(* Logix 5000 project; controller reports 1756-L63 rev 20.15; software revision 20.04 *)

TASK MainTask (continuous, watchdog 500 ms) : MainProgram, Report15Calcs, ReportCalcs

MODULES
   Local : 1756-L63 (ICP 0, rev 20.15)
END_MODULES

TYPE DateTime :
STRUCT
   Year : DINT;
   Month : DINT;
   Day : DINT;
   Hour : DINT;
   Minute : DINT;
   Second : DINT;
   Microsecond : DINT;   // Microsecond
   DayOfWeek : DINT;   // Day of week (Sunday = 0, Saturday = 6)
   DST_ON : BOOL;   // Day light Savings Time ON
END_STRUCT
END_TYPE

TYPE LogPoint :
STRUCT
   min : REAL;
   max : REAL;
   total : REAL;
   time : REAL;
   minminute : DINT;
   maxminute : DINT;
   valid : BOOL;
END_STRUCT
END_TYPE

TYPE LogRecord :
STRUCT
   log_data : LogPoint[125];
   time : DateTime;
END_STRUCT
END_TYPE

TYPE LogRecord15 :
STRUCT
   log_data : LogPoint[20];
   time : DateTime;
END_STRUCT
END_TYPE

TYPE LogRecord5 :
STRUCT
   log_data : LogPoint[20];
   time : DateTime;
END_STRUCT
END_TYPE

TYPE MOTOR :
STRUCT
   fail_dlay : DINT;
   mode_dlay : DINT;
   start_dlay : DINT;
   auto : BOOL;
   stop_man : BOOL;
   start_man : BOOL;
   fail_reset : BOOL;
   remote : BOOL;
   permit : BOOL;
   stop_sts : BOOL;
   run_sts : BOOL;
   stop_auto : BOOL;
   start_auto : BOOL;
   stop_out : BOOL;
   start_out : BOOL;
   run_out : BOOL;
   fail : BOOL;
   runtime : REAL;
   log : BOOL;
   Gen_Alarm : BOOL;   // General Alarm
   runtime_f : REAL;
   runtime_i : DINT;
   fail_tonr : FBD_TIMER;
   start_os : FBD_ONESHOT;
   manual_mode_timer : FBD_TIMER;
END_STRUCT
END_TYPE

TYPE PRANALOG :
STRUCT
   MinEU : REAL;
   MaxEU : REAL;
   almdb : REAL;
   lag : REAL;
   calib : BOOL;
   hihilim : REAL;
   hilim : REAL;
   lolim : REAL;
   lololim : REAL;
   raw : REAL;
   hold : BOOL;
   calc : REAL;
   value : REAL;
   valid : BOOL;
   log : BOOL;
   hihiraw : BOOL;
   hiraw : BOOL;
   loraw : BOOL;
   loloraw : BOOL;
END_STRUCT
END_TYPE

VAR_GLOBAL   (* controller tags *)
   AIT501do : PRANALOG := (MaxEU := 10.0, hihilim := 10.0, hilim := 8.0, lolim := 0.5, lololim := 0.5, raw := 21.951172, calc := 0.021951173, value := 0.021951173, valid := 1, log := 1, loraw := 1, loloraw := 1);   // Aeration tank 1 DO
   AIT501ph : PRANALOG := (MaxEU := 14.0, hihilim := 8.5, hilim := 8.0, lolim := 6.5, lololim := 6.3, raw := 5438.2197, calc := 7.6135077, value := 7.6135077, valid := 1, log := 1);   // Aeration tank 1 pH
   AIT502do : PRANALOG := (MaxEU := 10.0, hihilim := 10.0, hilim := 8.0, lolim := 0.5, lololim := 0.3, raw := 9517.547, calc := 9.517547, value := 9.517547, valid := 1, log := 1, hiraw := 1);   // Aeration tank 2 DO
   AIT502ph : PRANALOG := (MaxEU := 14.0, hihilim := 8.5, hilim := 8.0, lolim := 6.5, lololim := 6.3, raw := 4820.0977, calc := 6.7481365, value := 6.7481365, valid := 1, log := 1);   // Aeration tank 2 pH
   B301 : MOTOR := (fail_dlay := 60, start_dlay := 3000, permit := 1, run_sts := 1, runtime := 22541.49, runtime_f := 0.48989543, runtime_i := 22541, fail_tonr.TimerEnable := 1, fail_tonr.PRE := 60000, fail_tonr.Reset := 1, manual_mode_timer.Reset := 1);   // Equalization blower 1
   B302 : MOTOR := (fail_dlay := 60, start_dlay := 3000, permit := 1, run_sts := 1, runtime := 22540.76, runtime_f := 0.7594519, runtime_i := 22540, fail_tonr.TimerEnable := 1, fail_tonr.PRE := 60000, fail_tonr.Reset := 1, manual_mode_timer.Reset := 1);   // Equalization blower 2
   B303 : MOTOR := (fail_dlay := 60, start_dlay := 3000, permit := 1, stop_sts := 1, runtime := 0.2709657, runtime_f := 0.2709657, fail_tonr.TimerEnable := 1, fail_tonr.PRE := 60000, fail_tonr.Reset := 1, manual_mode_timer.Reset := 1);   // Equalization blower 3
   B501 : MOTOR := (fail_dlay := 60, start_dlay := 3000, auto := 1, remote := 1, permit := 1, stop_sts := 1, runtime := 10393.742, runtime_f := 0.7422347, runtime_i := 10393, fail_tonr.TimerEnable := 1, fail_tonr.PRE := 60000, fail_tonr.Reset := 1, manual_mode_timer.Reset := 1);   // Aeration tank 1 blower 1
   B502 : MOTOR := (fail_dlay := 60, start_dlay := 3000, auto := 1, remote := 1, permit := 1, stop_sts := 1, runtime := 6931.7354, runtime_f := 0.7353562, runtime_i := 6931, fail_tonr.TimerEnable := 1, fail_tonr.PRE := 60000, fail_tonr.Reset := 1, manual_mode_timer.Reset := 1);   // Aeration tank standby blower
   B503 : MOTOR := (fail_dlay := 60, start_dlay := 3000, auto := 1, remote := 1, permit := 1, run_sts := 1, run_out := 1, runtime := 5280.543, runtime_f := 0.5429669, runtime_i := 5280, fail_tonr.TimerEnable := 1, fail_tonr.PRE := 60000, fail_tonr.Reset := 1, start_os.InputBit := 1, manual_mode_timer.Reset := 1);   // Aeration tank 2 blower 1
   B601 : MOTOR := (fail_dlay := 60, start_dlay := 3000, remote := 1, permit := 1, stop_sts := 1, runtime := 17313.322, runtime_f := 0.32298738, runtime_i := 17313, fail_tonr.TimerEnable := 1, fail_tonr.PRE := 60000, fail_tonr.Reset := 1, manual_mode_timer.Reset := 1);   // Membrane tank 1 blower
   B602 : MOTOR := (fail_dlay := 60, start_dlay := 3000, remote := 1, permit := 1, stop_sts := 1, runtime := 12808.301, runtime_f := 0.30105218, runtime_i := 12808, fail_tonr.TimerEnable := 1, fail_tonr.PRE := 60000, fail_tonr.Reset := 1, manual_mode_timer.Reset := 1);   // Membrane tank 2 blower
   B603 : MOTOR := (fail_dlay := 60, start_dlay := 3000, auto := 1, remote := 1, permit := 1, run_sts := 1, run_out := 1, runtime := 5284.875, runtime_f := 0.87495077, runtime_i := 5284, fail_tonr.TimerEnable := 1, fail_tonr.PRE := 60000, fail_tonr.Reset := 1, start_os.InputBit := 1, manual_mode_timer.Reset := 1);   // Membrane tank 3 blower
   B604 : MOTOR := (fail_dlay := 60, start_dlay := 3000, auto := 1, remote := 1, permit := 1, run_sts := 1, run_out := 1, runtime := 5284.831, runtime_f := 0.8312785, runtime_i := 5284, fail_tonr.TimerEnable := 1, fail_tonr.PRE := 60000, fail_tonr.Reset := 1, start_os.InputBit := 1, manual_mode_timer.Reset := 1);   // Membrane tank 4 blower
   B901 : MOTOR := (fail_dlay := 60, start_dlay := 3000, remote := 1, permit := 1, stop_sts := 1, runtime := 1391.3846, runtime_f := 0.38459536, runtime_i := 1391, fail_tonr.TimerEnable := 1, fail_tonr.PRE := 60000, fail_tonr.Reset := 1, manual_mode_timer.Reset := 1);   // Digester blower 1
   B902 : MOTOR := (fail_dlay := 60, start_dlay := 3000, auto := 1, remote := 1, permit := 1, run_sts := 1, run_out := 1, runtime := 6851.961, runtime_f := 0.9611715, runtime_i := 6851, fail_tonr.TimerEnable := 1, fail_tonr.PRE := 60000, fail_tonr.Reset := 1, start_os.InputBit := 1, manual_mode_timer.Reset := 1);   // Digester blower 2
   DIESEL : MOTOR := (fail_dlay := 60, start_dlay := 3000, remote := 1, permit := 1, stop_sts := 1, fail_tonr.TimerEnable := 1, fail_tonr.PRE := 60000, fail_tonr.Reset := 1, manual_mode_timer.Reset := 1);   // Diesel generator
   FIT201 : PRANALOG := (MaxEU := 20.0, hihilim := 25.0, hilim := 20.0, raw := 3597.2026, calc := 7.194405, value := 7.194405, valid := 1, log := 1);   // Plant influent flow to screens
   FIT701 : PRANALOG := (MaxEU := 5.0, hihilim := 2.5, hilim := 2.0, lolim := 0.1, lololim := 0.1, raw := -9.0, valid := 1, log := 1, loraw := 1, loloraw := 1);   // Membrane tank 1 permeate flow
   FIT702 : PRANALOG := (MaxEU := 5.0, hihilim := 2.0, hilim := 1.8, lolim := 0.1, lololim := 0.1, raw := -4.0, valid := 1, log := 1, loraw := 1, loloraw := 1);   // Membrane tank 2 permeate flow
   FIT703 : PRANALOG := (MaxEU := 5.0, hihilim := 2.5, hilim := 2.0, lolim := 0.1, lololim := 0.1, raw := -4.0, valid := 1, log := 1, loraw := 1, loloraw := 1);   // Membrane tank 3 permeate flow
   FIT704 : PRANALOG := (MaxEU := 5.0, hihilim := 2.5, hilim := 2.0, raw := -6.0, valid := 1, log := 1);   // Membrane tank 4 permeate flow
   FIT801 : PRANALOG := (MaxEU := 5.0, raw := -1.0, valid := 1, log := 1, hihiraw := 1, hiraw := 1);   // CIP flow
   FIT901 : PRANALOG := (MaxEU := 5.0, raw := -4.0, valid := 1, log := 1, hihiraw := 1, hiraw := 1);   // Membrane tanks 1 & 2 WAS flow
   FIT902 : PRANALOG := (MaxEU := 5.0, raw := -3.0, valid := 1, log := 1, hihiraw := 1, hiraw := 1);   // Membrane tanks 3 & 4 WAS flow
   FunctionBlock_Cycle_Time : REAL := 251.0;   // Main Task Cycle Time in mseconds
   GT7951 : PRANALOG := (hihilim := 12.0, hilim := 10.0, raw := 125.78931, valid := 1, log := 1);   // Screening area H2S monitor
   LIT302 : PRANALOG := (MaxEU := 6.0, hihilim := 3.0, hilim := 2.9, lolim := 0.2, lololim := 0.5, raw := 1689.8391, calc := 1.0139034, value := 1.0139034, valid := 1, log := 1);   // Equalization tank 302 Level
   LIT501 : PRANALOG := (MaxEU := 6.0, hihilim := 2.5, hilim := 3.0, lolim := 1.0, lololim := 1.5, raw := 3821.76, calc := 2.293056, value := 2.293056, valid := 1, log := 1);   // Aeration tank 1 Level
   LIT502 : PRANALOG := (MaxEU := 6.0, hihilim := 2.5, hilim := 3.0, lolim := 1.0, lololim := 1.5, raw := 3509.0679, calc := 2.1054406, value := 2.1054406, valid := 1, log := 1);   // Aeration tank 2 Level
   LIT6101 : PRANALOG := (MaxEU := 2.0, raw := 795.14307, calc := 0.15902862, value := 0.15902862, valid := 1, log := 1, hihiraw := 1, hiraw := 1);   // Coagulant tank 6101 level
   LIT6102 : PRANALOG := (MaxEU := 2.0, raw := 931.36914, calc := 0.18627383, value := 0.18627383, valid := 1, log := 1, hihiraw := 1, hiraw := 1);   // Caustic tank 6102 Leve
   P301 : MOTOR := (fail_dlay := 60, start_dlay := 3000, remote := 1, permit := 1, stop_sts := 1, runtime := 502.63425, runtime_f := 0.6342328, runtime_i := 502, fail_tonr.TimerEnable := 1, fail_tonr.PRE := 60000, fail_tonr.Reset := 1, manual_mode_timer.Reset := 1);   // Equalization pump 1
   P302 : MOTOR := (fail_dlay := 60, start_dlay := 3000, remote := 1, permit := 1, stop_sts := 1, runtime := 1.2261261, runtime_f := 0.22612606, runtime_i := 1, fail_tonr.TimerEnable := 1, fail_tonr.PRE := 60000, fail_tonr.Reset := 1, manual_mode_timer.Reset := 1);   // Equalization pump 2
   P303 : MOTOR := (fail_dlay := 60, start_dlay := 3000, auto := 1, remote := 1, permit := 1, stop_sts := 1, runtime := 201.53206, runtime_f := 0.5320589, runtime_i := 201, fail_tonr.TimerEnable := 1, fail_tonr.PRE := 60000, fail_tonr.Reset := 1, manual_mode_timer.Reset := 1);   // Equalization pump 3
   P501 : MOTOR := (fail_dlay := 60, start_dlay := 3000, remote := 1, permit := 1, stop_sts := 1, runtime := 14554.279, runtime_f := 0.27947924, runtime_i := 14554, fail_tonr.TimerEnable := 1, fail_tonr.PRE := 60000, fail_tonr.Reset := 1, manual_mode_timer.Reset := 1);   // Membrane tank 1 mixed liquor pump
   P502 : MOTOR := (fail_dlay := 60, start_dlay := 3000, remote := 1, permit := 1, stop_sts := 1, runtime := 11217.086, runtime_f := 0.08595178, runtime_i := 11217, fail_tonr.TimerEnable := 1, fail_tonr.PRE := 60000, fail_tonr.Reset := 1, manual_mode_timer.Reset := 1);   // Membrane tank 2 mixed liquor pump
   P503 : MOTOR := (fail_dlay := 60, start_dlay := 3000, auto := 1, remote := 1, permit := 1, stop_sts := 1, runtime := 4799.387, runtime_f := 0.38708004, runtime_i := 4799, fail_tonr.TimerEnable := 1, fail_tonr.PRE := 60000, fail_tonr.Reset := 1, manual_mode_timer.Reset := 1);   // Membrane tank 3 mixed liquor pump
   P504 : MOTOR := (fail_dlay := 60, start_dlay := 3000, auto := 1, remote := 1, permit := 1, stop_sts := 1, runtime := 4738.982, runtime_f := 0.98173386, runtime_i := 4738, fail_tonr.TimerEnable := 1, fail_tonr.PRE := 60000, fail_tonr.Reset := 1, manual_mode_timer.Reset := 1);   // Membrane tank 4 mixed liquor pump
   P7011 : MOTOR := (fail_dlay := 60, start_dlay := 3000, auto := 1, remote := 1, permit := 1, stop_sts := 1, runtime := 6253.749, runtime_f := 0.7490861, runtime_i := 6253, fail_tonr.TimerEnable := 1, fail_tonr.PRE := 60000, fail_tonr.Reset := 1, manual_mode_timer.Reset := 1);   // Membrane tank 1 permeate pump 1
   P7012 : MOTOR := (fail_dlay := 60, start_dlay := 3000, auto := 1, remote := 1, permit := 1, stop_sts := 1, runtime := 5870.5024, runtime_f := 0.502557, runtime_i := 5870, fail_tonr.TimerEnable := 1, fail_tonr.PRE := 60000, fail_tonr.Reset := 1, manual_mode_timer.Reset := 1);   // Membrane tank 1 permeate pump 2
   P7021 : MOTOR := (fail_dlay := 60, start_dlay := 3000, auto := 1, remote := 1, permit := 1, stop_sts := 1, runtime := 4789.597, runtime_f := 0.59710574, runtime_i := 4789, fail_tonr.TimerEnable := 1, fail_tonr.PRE := 60000, fail_tonr.Reset := 1, manual_mode_timer.Reset := 1);   // Membrane tank 2 permeate pump 1
   P7022 : MOTOR := (fail_dlay := 60, start_dlay := 3000, auto := 1, remote := 1, permit := 1, stop_sts := 1, runtime := 4792.9336, runtime_f := 0.9336782, runtime_i := 4792, fail_tonr.TimerEnable := 1, fail_tonr.PRE := 60000, fail_tonr.Reset := 1, manual_mode_timer.Reset := 1);   // Membrane tank 2 permeate pump 2
   P7031 : MOTOR := (fail_dlay := 60, start_dlay := 3000, auto := 1, remote := 1, permit := 1, stop_sts := 1, runtime := 2042.6858, runtime_f := 0.6858263, runtime_i := 2042, fail_tonr.TimerEnable := 1, fail_tonr.PRE := 60000, fail_tonr.Reset := 1, manual_mode_timer.Reset := 1);   // Membrane tank 3 permeate pump 1
   P7032 : MOTOR := (fail_dlay := 60, start_dlay := 3000, auto := 1, remote := 1, permit := 1, stop_sts := 1, runtime := 2005.9248, runtime_f := 0.924792, runtime_i := 2005, fail_tonr.TimerEnable := 1, fail_tonr.PRE := 60000, fail_tonr.Reset := 1, manual_mode_timer.Reset := 1);   // Membrane tank 3 permeate pump 2
   P7041 : MOTOR := (fail_dlay := 60, start_dlay := 3000, auto := 1, remote := 1, permit := 1, stop_sts := 1, runtime := 1973.3212, runtime_f := 0.32117462, runtime_i := 1973, fail_tonr.TimerEnable := 1, fail_tonr.PRE := 60000, fail_tonr.Reset := 1, manual_mode_timer.Reset := 1);   // Membrane tank 4 permeate pump 1
   P7042 : MOTOR := (fail_dlay := 60, start_dlay := 3000, auto := 1, remote := 1, permit := 1, stop_sts := 1, runtime := 1973.0812, runtime_f := 0.081213675, runtime_i := 1973, fail_tonr.TimerEnable := 1, fail_tonr.PRE := 60000, fail_tonr.Reset := 1, manual_mode_timer.Reset := 1);   // Membrane tank 4 permeate pump 2
   P7951 : MOTOR := (permit := 1, stop_sts := 1, fail_tonr.TimerEnable := 1, fail_tonr.Reset := 1, manual_mode_timer.Reset := 1);   // Screen building sump pump
   P801 : MOTOR := (fail_dlay := 60, start_dlay := 3000, auto := 1, remote := 1, permit := 1, stop_sts := 1, runtime := 62.99539, runtime_f := 0.9953907, runtime_i := 62, fail_tonr.TimerEnable := 1, fail_tonr.PRE := 60000, fail_tonr.Reset := 1, manual_mode_timer.Reset := 1);   // CIP pump 1
   P802 : MOTOR := (fail_dlay := 60, auto := 1, remote := 1, permit := 1, stop_sts := 1, runtime := 411.53458, runtime_f := 0.5345711, runtime_i := 411, fail_tonr.TimerEnable := 1, fail_tonr.PRE := 60000, fail_tonr.Reset := 1, manual_mode_timer.Reset := 1);   // CIP Pump 2
   P901 : MOTOR := (fail_dlay := 60, start_dlay := 3000, remote := 1, permit := 1, stop_sts := 1, runtime := 70.41078, runtime_f := 0.4107828, runtime_i := 70, fail_tonr.TimerEnable := 1, fail_tonr.PRE := 60000, fail_tonr.Reset := 1, manual_mode_timer.Reset := 1);   // Membrane tank 1 WAS pump
   P902 : MOTOR := (fail_dlay := 60, start_dlay := 3000, remote := 1, permit := 1, stop_sts := 1, runtime := 51.641758, runtime_f := 0.6417567, runtime_i := 51, fail_tonr.TimerEnable := 1, fail_tonr.PRE := 60000, fail_tonr.Reset := 1, manual_mode_timer.Reset := 1);   // Membrane tank 2 WAS pump
   P903 : MOTOR := (fail_dlay := 60, start_dlay := 3000, remote := 1, permit := 1, run_sts := 1, run_out := 1, runtime := 14599.742, runtime_f := 0.7419928, runtime_i := 14599, fail_tonr.TimerEnable := 1, fail_tonr.PRE := 60000, fail_tonr.Reset := 1, start_os.InputBit := 1, manual_mode_timer.Reset := 1);   // Digester decant pump
   P904 : MOTOR := (fail_dlay := 60, start_dlay := 3000, remote := 1, permit := 1, stop_sts := 1, runtime := 23.586103, runtime_f := 0.58610374, runtime_i := 23, fail_tonr.TimerEnable := 1, fail_tonr.PRE := 60000, fail_tonr.Reset := 1, manual_mode_timer.Reset := 1);   // Membrane tank 4 WAS pump
   P905 : MOTOR := (fail_dlay := 60, start_dlay := 3000, remote := 1, permit := 1, stop_sts := 1, runtime := 22.263817, runtime_f := 0.26381716, runtime_i := 22, fail_tonr.TimerEnable := 1, fail_tonr.PRE := 60000, fail_tonr.Reset := 1, manual_mode_timer.Reset := 1);   // Membrane tank 3 WAS pump
   report15_data : LogRecord15[800] := ([0].log_data[0].min := 1.0, [0].log_data[0].max := 1.0, [0].log_data[0].total := 900.0, [0].log_data[0].time := 900.0, [0].log_data[0].minminute := 15, [0].log_data[0].maxminute := 15, [0].log_data[0].valid := 1, [0].log_data[1].valid := 1, [0].log_data[2].valid := 1, [0].log_data[3].valid := 1, [0].log_data[4].valid := 1, [0].log_data[5].valid := 1, [0].log_data[6].valid := 1, [0].log_data[7].valid := 1, [0].log_data[8].valid := 1, [0].log_data[9].valid := 1, [0].log_data[10].valid := 1, [0].log_data[11].valid := 1, [0].log_data[12].valid := 1, [0].log_data[13].valid := 1, [0].log_data[14].valid := 1, [0].log_data[15].valid := 1, [0].log_data[16].valid := 1, [0].log_data[17].valid := 1, [0].log_data[18].valid := 1, [0].log_data[19].valid := 1, [0].time.Year := 2023, [0].time.Month := 1, [0].time.Day := 16, [0].time.Minute := 29, [0].time.Second := 59, [1].log_data[0].min := 1.0, [1].log_data[0].max := 1.0, [1].log_data[0].total := 900.0, [1].log_data[0].time := 900.0, [1].log_data[0].minminute := 30, [1].log_data[0].maxminute := 30, [1].log_data[0].valid := 1, [1].log_data[1].valid := 1, [1].log_data[2].valid := 1, [1].log_data[3].valid := 1, [1].log_data[4].valid := 1, [1].log_data[5].valid := 1, [1].log_data[6].valid := 1, [1].log_data[7].valid := 1, [1].log_data[8].valid := 1, [1].log_data[9].valid := 1, [1].log_data[10].valid := 1, [1].log_data[11].valid := 1, [1].log_data[12].valid := 1, [1].log_data[13].valid := 1, [1].log_data[14].valid := 1, [1].log_data[15].valid := 1, [1].log_data[16].valid := 1, [1].log_data[17].valid := 1, [1].log_data[18].valid := 1, [1].log_data[19].valid := 1, [1].time.Year := 2023, [1].time.Month := 1, [1].time.Day := 16,
        [1].time.Minute := 44, [1].time.Second := 59, [2].log_data[0].min := 1.0, [2].log_data[0].max := 1.0, [2].log_data[0].total := 900.0, [2].log_data[0].time := 900.0, [2].log_data[0].minminute := 45, [2].log_data[0].maxminute := 45, [2].log_data[0].valid := 1, [2].log_data[1].valid := 1, [2].log_data[2].valid := 1, [2].log_data[3].valid := 1, [2].log_data[4].valid := 1, [2].log_data[5].valid := 1, [2].log_data[6].valid := 1, [2].log_data[7].valid := 1, [2].log_data[8].valid := 1, [2].log_data[9].valid := 1, [2].log_data[10].valid := 1, [2].log_data[11].valid := 1, [2].log_data[12].valid := 1, [2].log_data[13].valid := 1, [2].log_data[14].valid := 1, [2].log_data[15].valid := 1, [2].log_data[16].valid := 1, [2].log_data[17].valid := 1, [2].log_data[18].valid := 1, [2].log_data[19].valid := 1, [2].time.Year := 2023, [2].time.Month := 1, [2].time.Day := 16, [2].time.Minute := 59, [2].time.Second := 59, [3].log_data[0].min := 1.0, [3].log_data[0].max := 1.0, [3].log_data[0].total := 900.0, [3].log_data[0].time := 900.0, [3].log_data[0].valid := 1, [3].log_data[1].valid := 1, [3].log_data[2].valid := 1, [3].log_data[3].valid := 1, [3].log_data[4].valid := 1, [3].log_data[5].valid := 1, [3].log_data[6].valid := 1, [3].log_data[7].valid := 1, [3].log_data[8].valid := 1, [3].log_data[9].valid := 1, [3].log_data[10].valid := 1, [3].log_data[11].valid := 1, [3].log_data[12].valid := 1, [3].log_data[13].valid := 1, [3].log_data[14].valid := 1, [3].log_data[15].valid := 1, [3].log_data[16].valid := 1, [3].log_data[17].valid := 1, [3].log_data[18].valid := 1, [3].log_data[19].valid := 1, [3].time.Year := 2023, [3].time.Month := 1, [3].time.Day := 16,
        [3].time.Hour := 1, [3].time.Minute := 14, [3].time.Second := 59, [4].log_data[0].min := 1.0, [4].log_data[0].max := 1.0, [4].log_data[0].total := 900.0, [4].log_data[0].time := 900.0, [4].log_data[0].minminute := 15, [4].log_data[0].maxminute := 15, [4].log_data[0].valid := 1, [4].log_data[1].valid := 1, [4].log_data[2].valid := 1, [4].log_data[3].valid := 1, [4].log_data[4].valid := 1, [4].log_data[5].valid := 1, [4].log_data[6].valid := 1, [4].log_data[7].valid := 1, [4].log_data[8].valid := 1, [4].log_data[9].valid := 1, [4].log_data[10].valid := 1, [4].log_data[11].valid := 1, [4].log_data[12].valid := 1, [4].log_data[13].valid := 1, [4].log_data[14].valid := 1, [4].log_data[15].valid := 1, [4].log_data[16].valid := 1, [4].log_data[17].valid := 1, [4].log_data[18].valid := 1, [4].log_data[19].valid := 1, [4].time.Year := 2023, [4].time.Month := 1, [4].time.Day := 16, [4].time.Hour := 1, [4].time.Minute := 29, [4].time.Second := 59, [5].log_data[0].min := 1.0, [5].log_data[0].max := 1.0, [5].log_data[0].total := 900.0, [5].log_data[0].time := 900.0, [5].log_data[0].minminute := 30, [5].log_data[0].maxminute := 30, [5].log_data[0].valid := 1, [5].log_data[1].valid := 1, [5].log_data[2].valid := 1, [5].log_data[3].valid := 1, [5].log_data[4].valid := 1, [5].log_data[5].valid := 1, [5].log_data[6].valid := 1, [5].log_data[7].valid := 1, [5].log_data[8].valid := 1, [5].log_data[9].valid := 1, [5].log_data[10].valid := 1, [5].log_data[11].valid := 1, [5].log_data[12].valid := 1, [5].log_data[13].valid := 1, [5].log_data[14].valid := 1, [5].log_data[15].valid := 1, [5].log_data[16].valid := 1, [5].log_data[17].valid := 1, [5].log_data[18].valid := 1,
        [5].log_data[19].valid := 1, [5].time.Year := 2023, [5].time.Month := 1, [5].time.Day := 16, [5].time.Hour := 1, [5].time.Minute := 44, [5].time.Second := 59, [6].log_data[0].min := 1.0, [6].log_data[0].max := 1.0, [6].log_data[0].total := 900.0, [6].log_data[0].time := 900.0, [6].log_data[0].minminute := 45, [6].log_data[0].maxminute := 45, [6].log_data[0].valid := 1, [6].log_data[1].valid := 1, [6].log_data[2].valid := 1, [6].log_data[3].valid := 1, [6].log_data[4].valid := 1, [6].log_data[5].valid := 1, [6].log_data[6].valid := 1, [6].log_data[7].valid := 1, [6].log_data[8].valid := 1, [6].log_data[9].valid := 1, [6].log_data[10].valid := 1, [6].log_data[11].valid := 1, [6].log_data[12].valid := 1, [6].log_data[13].valid := 1, [6].log_data[14].valid := 1, [6].log_data[15].valid := 1, [6].log_data[16].valid := 1, [6].log_data[17].valid := 1, [6].log_data[18].valid := 1, [6].log_data[19].valid := 1, [6].time.Year := 2023, [6].time.Month := 1, [6].time.Day := 16, [6].time.Hour := 1, [6].time.Minute := 59, [6].time.Second := 59, [7].log_data[0].min := 1.0, [7].log_data[0].max := 1.0, [7].log_data[0].total := 900.0, [7].log_data[0].time := 900.0, [7].log_data[0].valid := 1, [7].log_data[1].valid := 1, [7].log_data[2].valid := 1, [7].log_data[3].valid := 1, [7].log_data[4].valid := 1, [7].log_data[5].valid := 1, [7].log_data[6].valid := 1, [7].log_data[7].valid := 1, [7].log_data[8].valid := 1, [7].log_data[9].valid := 1, [7].log_data[10].valid := 1, [7].log_data[11].valid := 1, [7].log_data[12].valid := 1, [7].log_data[13].valid := 1, [7].log_data[14].valid := 1, [7].log_data[15].valid := 1, [7].log_data[16].valid := 1,
        [7].log_data[17].valid := 1, [7].log_data[18].valid := 1, [7].log_data[19].valid := 1, [7].time.Year := 2023, [7].time.Month := 1, [7].time.Day := 16, [7].time.Hour := 2, [7].time.Minute := 14, [7].time.Second := 59, [8].log_data[0].min := 1.0, [8].log_data[0].max := 1.0, [8].log_data[0].total := 900.0, [8].log_data[0].time := 900.0, [8].log_data[0].minminute := 15, [8].log_data[0].maxminute := 15, [8].log_data[0].valid := 1, [8].log_data[1].valid := 1, [8].log_data[2].valid := 1, [8].log_data[3].valid := 1, [8].log_data[4].valid := 1, [8].log_data[5].valid := 1, [8].log_data[6].valid := 1, [8].log_data[7].valid := 1, [8].log_data[8].valid := 1, [8].log_data[9].valid := 1, [8].log_data[10].valid := 1, [8].log_data[11].valid := 1, [8].log_data[12].valid := 1, [8].log_data[13].valid := 1, [8].log_data[14].valid := 1, [8].log_data[15].valid := 1, [8].log_data[16].valid := 1, [8].log_data[17].valid := 1, [8].log_data[18].valid := 1, [8].log_data[19].valid := 1, [8].time.Year := 2023, [8].time.Month := 1, [8].time.Day := 16, [8].time.Hour := 2, [8].time.Minute := 29, [8].time.Second := 59, [9].log_data[0].min := 1.0, [9].log_data[0].max := 1.0, [9].log_data[0].total := 900.0, [9].log_data[0].time := 900.0, [9].log_data[0].minminute := 30, [9].log_data[0].maxminute := 30, [9].log_data[0].valid := 1, [9].log_data[1].valid := 1, [9].log_data[2].valid := 1, [9].log_data[3].valid := 1, [9].log_data[4].valid := 1, [9].log_data[5].valid := 1, [9].log_data[6].valid := 1, [9].log_data[7].valid := 1, [9].log_data[8].valid := 1, [9].log_data[9].valid := 1, [9].log_data[10].valid := 1, [9].log_data[11].valid := 1, [9].log_data[12].valid := 1,
        [9].log_data[13].valid := 1, [9].log_data[14].valid := 1, [9].log_data[15].valid := 1, [9].log_data[16].valid := 1, [9].log_data[17].valid := 1, [9].log_data[18].valid := 1, [9].log_data[19].valid := 1, [9].time.Year := 2023, [9].time.Month := 1, [9].time.Day := 16, [9].time.Hour := 2, [9].time.Minute := 44, [9].time.Second := 59, [10].log_data[0].min := 1.0, [10].log_data[0].max := 1.0, [10].log_data[0].total := 900.0, [10].log_data[0].time := 900.0, [10].log_data[0].minminute := 45, [10].log_data[0].maxminute := 45, [10].log_data[0].valid := 1, [10].log_data[1].valid := 1, [10].log_data[2].valid := 1, [10].log_data[3].valid := 1, [10].log_data[4].valid := 1, [10].log_data[5].valid := 1, [10].log_data[6].valid := 1, [10].log_data[7].valid := 1, [10].log_data[8].valid := 1, [10].log_data[9].valid := 1, [10].log_data[10].valid := 1, [10].log_data[11].valid := 1, [10].log_data[12].valid := 1, [10].log_data[13].valid := 1, [10].log_data[14].valid := 1, [10].log_data[15].valid := 1, [10].log_data[16].valid := 1, [10].log_data[17].valid := 1, [10].log_data[18].valid := 1, [10].log_data[19].valid := 1, [10].time.Year := 2023, [10].time.Month := 1, [10].time.Day := 16, [10].time.Hour := 2, [10].time.Minute := 59, [10].time.Second := 59, [11].log_data[0].min := 1.0, [11].log_data[0].max := 1.0, [11].log_data[0].total := 900.0, [11].log_data[0].time := 900.0, [11].log_data[0].valid := 1, [11].log_data[1].valid := 1, [11].log_data[2].valid := 1, [11].log_data[3].valid := 1, [11].log_data[4].valid := 1, [11].log_data[5].valid := 1, [11].log_data[6].valid := 1, [11].log_data[7].valid := 1, [11].log_data[8].valid := 1, [11].log_data[9].valid := 1, [11].log_data[10].valid := 1,
        [11].log_data[11].valid := 1, [11].log_data[12].valid := 1, [11].log_data[13].valid := 1, [11].log_data[14].valid := 1, [11].log_data[15].valid := 1, [11].log_data[16].valid := 1, [11].log_data[17].valid := 1, [11].log_data[18].valid := 1, [11].log_data[19].valid := 1, [11].time.Year := 2023, [11].time.Month := 1, [11].time.Day := 16, [11].time.Hour := 3, [11].time.Minute := 14, [11].time.Second := 59, [12].log_data[0].min := 1.0, [12].log_data[0].max := 1.0, [12].log_data[0].total := 900.0, [12].log_data[0].time := 900.0, [12].log_data[0].minminute := 15, [12].log_data[0].maxminute := 15, [12].log_data[0].valid := 1, [12].log_data[1].valid := 1, [12].log_data[2].valid := 1, [12].log_data[3].valid := 1, [12].log_data[4].valid := 1, [12].log_data[5].valid := 1, [12].log_data[6].valid := 1, [12].log_data[7].valid := 1, [12].log_data[8].valid := 1, [12].log_data[9].valid := 1, [12].log_data[10].valid := 1, [12].log_data[11].valid := 1, [12].log_data[12].valid := 1, [12].log_data[13].valid := 1, [12].log_data[14].valid := 1, [12].log_data[15].valid := 1, [12].log_data[16].valid := 1, [12].log_data[17].valid := 1, [12].log_data[18].valid := 1, [12].log_data[19].valid := 1, [12].time.Year := 2023, [12].time.Month := 1, [12].time.Day := 16, [12].time.Hour := 3, [12].time.Minute := 29, [12].time.Second := 59, [13].log_data[0].min := 1.0, [13].log_data[0].max := 1.0, [13].log_data[0].total := 900.0, [13].log_data[0].time := 900.0, [13].log_data[0].minminute := 30, [13].log_data[0].maxminute := 30, [13].log_data[0].valid := 1, [13].log_data[1].valid := 1, [13].log_data[2].valid := 1, [13].log_data[3].valid := 1, [13].log_data[4].valid := 1, [13].log_data[5].valid := 1, [13].log_data[6].valid := 1,
        [13].log_data[7].valid := 1, [13].log_data[8].valid := 1, [13].log_data[9].valid := 1, [13].log_data[10].valid := 1, [13].log_data[11].valid := 1, [13].log_data[12].valid := 1, [13].log_data[13].valid := 1, [13].log_data[14].valid := 1, [13].log_data[15].valid := 1, [13].log_data[16].valid := 1, [13].log_data[17].valid := 1, [13].log_data[18].valid := 1, [13].log_data[19].valid := 1, [13].time.Year := 2023, [13].time.Month := 1, [13].time.Day := 16, [13].time.Hour := 3, [13].time.Minute := 44, [13].time.Second := 59, [14].log_data[0].min := 1.0, [14].log_data[0].max := 1.0, [14].log_data[0].total := 900.0, [14].log_data[0].time := 900.0, [14].log_data[0].minminute := 45, [14].log_data[0].maxminute := 45, [14].log_data[0].valid := 1, [14].log_data[1].valid := 1, [14].log_data[2].valid := 1, [14].log_data[3].valid := 1, [14].log_data[4].valid := 1, [14].log_data[5].valid := 1, [14].log_data[6].valid := 1, [14].log_data[7].valid := 1, [14].log_data[8].valid := 1, [14].log_data[9].valid := 1, [14].log_data[10].valid := 1, [14].log_data[11].valid := 1, [14].log_data[12].valid := 1, [14].log_data[13].valid := 1, [14].log_data[14].valid := 1, [14].log_data[15].valid := 1, [14].log_data[16].valid := 1, [14].log_data[17].valid := 1, [14].log_data[18].valid := 1, [14].log_data[19].valid := 1, [14].time.Year := 2023, [14].time.Month := 1, [14].time.Day := 16, [14].time.Hour := 3, [14].time.Minute := 59, [14].time.Second := 59, [15].log_data[0].min := 1.0, [15].log_data[0].max := 1.0, [15].log_data[0].total := 900.0, [15].log_data[0].time := 900.0, [15].log_data[0].valid := 1, [15].log_data[1].valid := 1, [15].log_data[2].valid := 1, [15].log_data[3].valid := 1, [15].log_data[4].valid := 1,
        [15].log_data[5].valid := 1, [15].log_data[6].valid := 1, [15].log_data[7].valid := 1, [15].log_data[8].valid := 1, [15].log_data[9].valid := 1, [15].log_data[10].valid := 1, [15].log_data[11].valid := 1, [15].log_data[12].valid := 1, [15].log_data[13].valid := 1, [15].log_data[14].valid := 1, [15].log_data[15].valid := 1, [15].log_data[16].valid := 1, [15].log_data[17].valid := 1, [15].log_data[18].valid := 1, [15].log_data[19].valid := 1, [15].time.Year := 2023, [15].time.Month := 1, [15].time.Day := 16, [15].time.Hour := 4, [15].time.Minute := 14, [15].time.Second := 59, [16].log_data[0].min := 1.0, [16].log_data[0].max := 1.0, [16].log_data[0].total := 900.0, [16].log_data[0].time := 900.0, [16].log_data[0].minminute := 15, [16].log_data[0].maxminute := 15, [16].log_data[0].valid := 1, [16].log_data[1].valid := 1, [16].log_data[2].valid := 1, [16].log_data[3].valid := 1, [16].log_data[4].valid := 1, [16].log_data[5].valid := 1, [16].log_data[6].valid := 1, [16].log_data[7].valid := 1, [16].log_data[8].valid := 1, [16].log_data[9].valid := 1, [16].log_data[10].valid := 1, [16].log_data[11].valid := 1, [16].log_data[12].valid := 1, [16].log_data[13].valid := 1, [16].log_data[14].valid := 1, [16].log_data[15].valid := 1, [16].log_data[16].valid := 1, [16].log_data[17].valid := 1, [16].log_data[18].valid := 1, [16].log_data[19].valid := 1, [16].time.Year := 2023, [16].time.Month := 1, [16].time.Day := 16, [16].time.Hour := 4, [16].time.Minute := 29, [16].time.Second := 59, [17].log_data[0].min := 1.0, [17].log_data[0].max := 1.0, [17].log_data[0].total := 900.0, [17].log_data[0].time := 900.0, [17].log_data[0].minminute := 30, [17].log_data[0].maxminute := 30, [17].log_data[0].valid := 1,
        [17].log_data[1].valid := 1, [17].log_data[2].valid := 1, [17].log_data[3].valid := 1, [17].log_data[4].valid := 1, [17].log_data[5].valid := 1, [17].log_data[6].valid := 1, [17].log_data[7].valid := 1, [17].log_data[8].valid := 1, [17].log_data[9].valid := 1, [17].log_data[10].valid := 1, [17].log_data[11].valid := 1, [17].log_data[12].valid := 1, [17].log_data[13].valid := 1, [17].log_data[14].valid := 1, [17].log_data[15].valid := 1, [17].log_data[16].valid := 1, [17].log_data[17].valid := 1, [17].log_data[18].valid := 1, [17].log_data[19].valid := 1, [17].time.Year := 2023, [17].time.Month := 1, [17].time.Day := 16, [17].time.Hour := 4, [17].time.Minute := 44, [17].time.Second := 59, [18].log_data[0].min := 1.0, [18].log_data[0].max := 1.0, [18].log_data[0].total := 900.0, [18].log_data[0].time := 900.0, [18].log_data[0].minminute := 45, [18].log_data[0].maxminute := 45, [18].log_data[0].valid := 1, [18].log_data[1].valid := 1, [18].log_data[2].valid := 1, [18].log_data[3].valid := 1, [18].log_data[4].valid := 1, [18].log_data[5].valid := 1, [18].log_data[6].valid := 1, [18].log_data[7].valid := 1, [18].log_data[8].valid := 1, [18].log_data[9].valid := 1, [18].log_data[10].valid := 1, [18].log_data[11].valid := 1, [18].log_data[12].valid := 1, [18].log_data[13].valid := 1, [18].log_data[14].valid := 1, [18].log_data[15].valid := 1, [18].log_data[16].valid := 1, [18].log_data[17].valid := 1, [18].log_data[18].valid := 1, [18].log_data[19].valid := 1, [18].time.Year := 2023, [18].time.Month := 1, [18].time.Day := 16, [18].time.Hour := 4, [18].time.Minute := 59, [18].time.Second := 59, [19].log_data[0].min := 1.0, [19].log_data[0].max := 1.0, [19].log_data[0].total := 900.0,
        [19].log_data[0].time := 900.0, [19].log_data[0].valid := 1, [19].log_data[1].valid := 1, [19].log_data[2].valid := 1, [19].log_data[3].valid := 1, [19].log_data[4].valid := 1, [19].log_data[5].valid := 1, [19].log_data[6].valid := 1, [19].log_data[7].valid := 1, [19].log_data[8].valid := 1, [19].log_data[9].valid := 1, [19].log_data[10].valid := 1, [19].log_data[11].valid := 1, [19].log_data[12].valid := 1, [19].log_data[13].valid := 1, [19].log_data[14].valid := 1, [19].log_data[15].valid := 1, [19].log_data[16].valid := 1, [19].log_data[17].valid := 1, [19].log_data[18].valid := 1, [19].log_data[19].valid := 1, [19].time.Year := 2023, [19].time.Month := 1, [19].time.Day := 16, [19].time.Hour := 5, [19].time.Minute := 14, [19].time.Second := 59, [20].log_data[0].min := 1.0, [20].log_data[0].max := 1.0, [20].log_data[0].total := 900.0, [20].log_data[0].time := 900.0, [20].log_data[0].minminute := 15, [20].log_data[0].maxminute := 15, [20].log_data[0].valid := 1, [20].log_data[1].valid := 1, [20].log_data[2].valid := 1, [20].log_data[3].valid := 1, [20].log_data[4].valid := 1, [20].log_data[5].valid := 1, [20].log_data[6].valid := 1, [20].log_data[7].valid := 1, [20].log_data[8].valid := 1, [20].log_data[9].valid := 1, [20].log_data[10].valid := 1, [20].log_data[11].valid := 1, [20].log_data[12].valid := 1, [20].log_data[13].valid := 1, [20].log_data[14].valid := 1, [20].log_data[15].valid := 1, [20].log_data[16].valid := 1, [20].log_data[17].valid := 1, [20].log_data[18].valid := 1, [20].log_data[19].valid := 1, [20].time.Year := 2023, [20].time.Month := 1, [20].time.Day := 16, [20].time.Hour := 5, [20].time.Minute := 29, [20].time.Second := 59, [21].log_data[0].min := 1.0,
        [21].log_data[0].max := 1.0, [21].log_data[0].total := 900.0, [21].log_data[0].time := 900.0, [21].log_data[0].minminute := 30, [21].log_data[0].maxminute := 30, [21].log_data[0].valid := 1, [21].log_data[1].valid := 1, [21].log_data[2].valid := 1, [21].log_data[3].valid := 1, [21].log_data[4].valid := 1, [21].log_data[5].valid := 1, [21].log_data[6].valid := 1, [21].log_data[7].valid := 1, [21].log_data[8].valid := 1, [21].log_data[9].valid := 1, [21].log_data[10].valid := 1, [21].log_data[11].valid := 1, [21].log_data[12].valid := 1, [21].log_data[13].valid := 1, [21].log_data[14].valid := 1, [21].log_data[15].valid := 1, [21].log_data[16].valid := 1, [21].log_data[17].valid := 1, [21].log_data[18].valid := 1, [21].log_data[19].valid := 1, [21].time.Year := 2023, [21].time.Month := 1, [21].time.Day := 16, [21].time.Hour := 5, [21].time.Minute := 44, [21].time.Second := 59, [22].log_data[0].min := 1.0, [22].log_data[0].max := 1.0, [22].log_data[0].total := 900.0, [22].log_data[0].time := 900.0, [22].log_data[0].minminute := 45, [22].log_data[0].maxminute := 45, [22].log_data[0].valid := 1, [22].log_data[1].valid := 1, [22].log_data[2].valid := 1, [22].log_data[3].valid := 1, [22].log_data[4].valid := 1, [22].log_data[5].valid := 1, [22].log_data[6].valid := 1, [22].log_data[7].valid := 1, [22].log_data[8].valid := 1, [22].log_data[9].valid := 1, [22].log_data[10].valid := 1, [22].log_data[11].valid := 1, [22].log_data[12].valid := 1, [22].log_data[13].valid := 1, [22].log_data[14].valid := 1, [22].log_data[15].valid := 1, [22].log_data[16].valid := 1, [22].log_data[17].valid := 1, [22].log_data[18].valid := 1, [22].log_data[19].valid := 1, [22].time.Year := 2023, [22].time.Month := 1, [22].time.Day := 16,
        [22].time.Hour := 5, [22].time.Minute := 59, [22].time.Second := 59, [23].log_data[0].min := 1.0, [23].log_data[0].max := 1.0, [23].log_data[0].total := 900.0, [23].log_data[0].time := 900.0, [23].log_data[0].valid := 1, [23].log_data[1].valid := 1, [23].log_data[2].valid := 1, [23].log_data[3].valid := 1, [23].log_data[4].valid := 1, [23].log_data[5].valid := 1, [23].log_data[6].valid := 1, [23].log_data[7].valid := 1, [23].log_data[8].valid := 1, [23].log_data[9].valid := 1, [23].log_data[10].valid := 1, [23].log_data[11].valid := 1, [23].log_data[12].valid := 1, [23].log_data[13].valid := 1, [23].log_data[14].valid := 1, [23].log_data[15].valid := 1, [23].log_data[16].valid := 1, [23].log_data[17].valid := 1, [23].log_data[18].valid := 1, [23].log_data[19].valid := 1, [23].time.Year := 2023, [23].time.Month := 1, [23].time.Day := 16, [23].time.Hour := 6, [23].time.Minute := 14, [23].time.Second := 59, [24].log_data[0].min := 1.0, [24].log_data[0].max := 1.0, [24].log_data[0].total := 900.0, [24].log_data[0].time := 900.0, [24].log_data[0].minminute := 15, [24].log_data[0].maxminute := 15, [24].log_data[0].valid := 1, [24].log_data[1].valid := 1, [24].log_data[2].valid := 1, [24].log_data[3].valid := 1, [24].log_data[4].valid := 1, [24].log_data[5].valid := 1, [24].log_data[6].valid := 1, [24].log_data[7].valid := 1, [24].log_data[8].valid := 1, [24].log_data[9].valid := 1, [24].log_data[10].valid := 1, [24].log_data[11].valid := 1, [24].log_data[12].valid := 1, [24].log_data[13].valid := 1, [24].log_data[14].valid := 1, [24].log_data[15].valid := 1, [24].log_data[16].valid := 1, [24].log_data[17].valid := 1, [24].log_data[18].valid := 1, [24].log_data[19].valid := 1, [24].time.Year := 2023,
        [24].time.Month := 1, [24].time.Day := 16, [24].time.Hour := 6, [24].time.Minute := 29, [24].time.Second := 59, [25].log_data[0].min := 1.0, [25].log_data[0].max := 1.0, [25].log_data[0].total := 900.0, [25].log_data[0].time := 900.0, [25].log_data[0].minminute := 30, [25].log_data[0].maxminute := 30, [25].log_data[0].valid := 1, [25].log_data[1].valid := 1, [25].log_data[2].valid := 1, [25].log_data[3].valid := 1, [25].log_data[4].valid := 1, [25].log_data[5].valid := 1, [25].log_data[6].valid := 1, [25].log_data[7].valid := 1, [25].log_data[8].valid := 1, [25].log_data[9].valid := 1, [25].log_data[10].valid := 1, [25].log_data[11].valid := 1, [25].log_data[12].valid := 1, [25].log_data[13].valid := 1, [25].log_data[14].valid := 1, [25].log_data[15].valid := 1, [25].log_data[16].valid := 1, [25].log_data[17].valid := 1, [25].log_data[18].valid := 1, [25].log_data[19].valid := 1, [25].time.Year := 2023, [25].time.Month := 1, [25].time.Day := 16, [25].time.Hour := 6, [25].time.Minute := 44, [25].time.Second := 59, [26].log_data[0].min := 1.0, [26].log_data[0].max := 1.0, [26].log_data[0].total := 900.0, [26].log_data[0].time := 900.0, [26].log_data[0].minminute := 45, [26].log_data[0].maxminute := 45, [26].log_data[0].valid := 1, [26].log_data[1].valid := 1, [26].log_data[2].valid := 1, [26].log_data[3].valid := 1, [26].log_data[4].valid := 1, [26].log_data[5].valid := 1, [26].log_data[6].valid := 1, [26].log_data[7].valid := 1, [26].log_data[8].valid := 1, [26].log_data[9].valid := 1, [26].log_data[10].valid := 1, [26].log_data[11].valid := 1, [26].log_data[12].valid := 1, [26].log_data[13].valid := 1, [26].log_data[14].valid := 1, [26].log_data[15].valid := 1, [26].log_data[16].valid := 1,
        [26].log_data[17].valid := 1, [26].log_data[18].valid := 1, [26].log_data[19].valid := 1, [26].time.Year := 2023, [26].time.Month := 1, [26].time.Day := 16, [26].time.Hour := 6, [26].time.Minute := 59, [26].time.Second := 59, [27].log_data[0].min := 1.0, [27].log_data[0].max := 1.0, [27].log_data[0].total := 900.0, [27].log_data[0].time := 900.0, [27].log_data[0].valid := 1, [27].log_data[1].valid := 1, [27].log_data[2].valid := 1, [27].log_data[3].valid := 1, [27].log_data[4].valid := 1, [27].log_data[5].valid := 1, [27].log_data[6].valid := 1, [27].log_data[7].valid := 1, [27].log_data[8].valid := 1, [27].log_data[9].valid := 1, [27].log_data[10].valid := 1, [27].log_data[11].valid := 1, [27].log_data[12].valid := 1, [27].log_data[13].valid := 1, [27].log_data[14].valid := 1, [27].log_data[15].valid := 1, [27].log_data[16].valid := 1, [27].log_data[17].valid := 1, [27].log_data[18].valid := 1, [27].log_data[19].valid := 1, [27].time.Year := 2023, [27].time.Month := 1, [27].time.Day := 16, [27].time.Hour := 7, [27].time.Minute := 14, [27].time.Second := 59, [28].log_data[0].min := 1.0, [28].log_data[0].max := 1.0, [28].log_data[0].total := 900.0, [28].log_data[0].time := 900.0, [28].log_data[0].minminute := 15, [28].log_data[0].maxminute := 15, [28].log_data[0].valid := 1, [28].log_data[1].valid := 1, [28].log_data[2].valid := 1, [28].log_data[3].valid := 1, [28].log_data[4].valid := 1, [28].log_data[5].valid := 1, [28].log_data[6].valid := 1, [28].log_data[7].valid := 1, [28].log_data[8].valid := 1, [28].log_data[9].valid := 1, [28].log_data[10].valid := 1, [28].log_data[11].valid := 1, [28].log_data[12].valid := 1, [28].log_data[13].valid := 1, [28].log_data[14].valid := 1,
        [28].log_data[15].valid := 1, [28].log_data[16].valid := 1, [28].log_data[17].valid := 1, [28].log_data[18].valid := 1, [28].log_data[19].valid := 1, [28].time.Year := 2023, [28].time.Month := 1, [28].time.Day := 16, [28].time.Hour := 7, [28].time.Minute := 29, [28].time.Second := 59, [29].log_data[0].min := 1.0, [29].log_data[0].max := 1.0, [29].log_data[0].total := 900.0, [29].log_data[0].time := 900.0, [29].log_data[0].minminute := 30, [29].log_data[0].maxminute := 30, [29].log_data[0].valid := 1, [29].log_data[1].valid := 1, [29].log_data[2].valid := 1, [29].log_data[3].valid := 1, [29].log_data[4].valid := 1, [29].log_data[5].valid := 1, [29].log_data[6].valid := 1, [29].log_data[7].valid := 1, [29].log_data[8].valid := 1, [29].log_data[9].valid := 1, [29].log_data[10].valid := 1, [29].log_data[11].valid := 1, [29].log_data[12].valid := 1, [29].log_data[13].valid := 1, [29].log_data[14].valid := 1, [29].log_data[15].valid := 1, [29].log_data[16].valid := 1, [29].log_data[17].valid := 1, [29].log_data[18].valid := 1, [29].log_data[19].valid := 1, [29].time.Year := 2023, [29].time.Month := 1, [29].time.Day := 16, [29].time.Hour := 7, [29].time.Minute := 44, [29].time.Second := 59, [30].log_data[0].min := 1.0, [30].log_data[0].max := 1.0, [30].log_data[0].total := 900.0, [30].log_data[0].time := 900.0, [30].log_data[0].minminute := 45, [30].log_data[0].maxminute := 45, [30].log_data[0].valid := 1, [30].log_data[1].valid := 1, [30].log_data[2].valid := 1, [30].log_data[3].valid := 1, [30].log_data[4].valid := 1, [30].log_data[5].valid := 1, [30].log_data[6].valid := 1, [30].log_data[7].valid := 1, [30].log_data[8].valid := 1, [30].log_data[9].valid := 1, [30].log_data[10].valid := 1,
        [30].log_data[11].valid := 1, [30].log_data[12].valid := 1, [30].log_data[13].valid := 1, [30].log_data[14].valid := 1, [30].log_data[15].valid := 1, [30].log_data[16].valid := 1, [30].log_data[17].valid := 1, [30].log_data[18].valid := 1, [30].log_data[19].valid := 1, [30].time.Year := 2023, [30].time.Month := 1, [30].time.Day := 16, [30].time.Hour := 7, [30].time.Minute := 59, [30].time.Second := 59, [31].log_data[0].min := 1.0, [31].log_data[0].max := 1.0, [31].log_data[0].total := 900.0, [31].log_data[0].time := 900.0, [31].log_data[0].valid := 1, [31].log_data[1].valid := 1, [31].log_data[2].valid := 1, [31].log_data[3].valid := 1, [31].log_data[4].valid := 1, [31].log_data[5].valid := 1, [31].log_data[6].valid := 1, [31].log_data[7].valid := 1, [31].log_data[8].valid := 1, [31].log_data[9].valid := 1, [31].log_data[10].valid := 1, [31].log_data[11].valid := 1, [31].log_data[12].valid := 1, [31].log_data[13].valid := 1, [31].log_data[14].valid := 1, [31].log_data[15].valid := 1, [31].log_data[16].valid := 1, [31].log_data[17].valid := 1, [31].log_data[18].valid := 1, [31].log_data[19].valid := 1, [31].time.Year := 2023, [31].time.Month := 1, [31].time.Day := 16, [31].time.Hour := 8, [31].time.Minute := 14, [31].time.Second := 59, [32].log_data[0].min := 1.0, [32].log_data[0].max := 1.0, [32].log_data[0].total := 900.0, [32].log_data[0].time := 900.0, [32].log_data[0].minminute := 15, [32].log_data[0].maxminute := 15, [32].log_data[0].valid := 1, [32].log_data[1].valid := 1, [32].log_data[2].valid := 1, [32].log_data[3].valid := 1, [32].log_data[4].valid := 1, [32].log_data[5].valid := 1, [32].log_data[6].valid := 1, [32].log_data[7].valid := 1, [32].log_data[8].valid := 1,
        [32].log_data[9].valid := 1, [32].log_data[10].valid := 1, [32].log_data[11].valid := 1, [32].log_data[12].valid := 1, [32].log_data[13].valid := 1, [32].log_data[14].valid := 1, [32].log_data[15].valid := 1, [32].log_data[16].valid := 1, [32].log_data[17].valid := 1, [32].log_data[18].valid := 1, [32].log_data[19].valid := 1, [32].time.Year := 2023, [32].time.Month := 1, [32].time.Day := 16, [32].time.Hour := 8, [32].time.Minute := 29, [32].time.Second := 59, [33].log_data[0].min := 1.0, [33].log_data[0].max := 1.0, [33].log_data[0].total := 900.0, [33].log_data[0].time := 900.0, [33].log_data[0].minminute := 30, [33].log_data[0].maxminute := 30, [33].log_data[0].valid := 1, [33].log_data[1].valid := 1, [33].log_data[2].valid := 1, [33].log_data[3].valid := 1, [33].log_data[4].valid := 1, [33].log_data[5].valid := 1, [33].log_data[6].valid := 1, [33].log_data[7].valid := 1, [33].log_data[8].valid := 1, [33].log_data[9].valid := 1, [33].log_data[10].valid := 1, [33].log_data[11].valid := 1, [33].log_data[12].valid := 1, [33].log_data[13].valid := 1, [33].log_data[14].valid := 1, [33].log_data[15].valid := 1, [33].log_data[16].valid := 1, [33].log_data[17].valid := 1, [33].log_data[18].valid := 1, [33].log_data[19].valid := 1, [33].time.Year := 2023, [33].time.Month := 1, [33].time.Day := 16, [33].time.Hour := 8, [33].time.Minute := 44, [33].time.Second := 59, [34].log_data[0].min := 1.0, [34].log_data[0].max := 1.0, [34].log_data[0].total := 900.0, [34].log_data[0].time := 900.0, [34].log_data[0].minminute := 45, [34].log_data[0].maxminute := 45, [34].log_data[0].valid := 1, [34].log_data[1].valid := 1, [34].log_data[2].valid := 1, [34].log_data[3].valid := 1, [34].log_data[4].valid := 1,
        [34].log_data[5].valid := 1, [34].log_data[6].valid := 1, [34].log_data[7].valid := 1, [34].log_data[8].valid := 1, [34].log_data[9].valid := 1, [34].log_data[10].valid := 1, [34].log_data[11].valid := 1, [34].log_data[12].valid := 1, [34].log_data[13].valid := 1, [34].log_data[14].valid := 1, [34].log_data[15].valid := 1, [34].log_data[16].valid := 1, [34].log_data[17].valid := 1, [34].log_data[18].valid := 1, [34].log_data[19].valid := 1, [34].time.Year := 2023, [34].time.Month := 1, [34].time.Day := 16, [34].time.Hour := 8, [34].time.Minute := 59, [34].time.Second := 59, [35].log_data[0].min := 1.0, [35].log_data[0].max := 1.0, [35].log_data[0].total := 900.0, [35].log_data[0].time := 900.0, [35].log_data[0].valid := 1, [35].log_data[1].valid := 1, [35].log_data[2].valid := 1, [35].log_data[3].valid := 1, [35].log_data[4].valid := 1, [35].log_data[5].valid := 1, [35].log_data[6].valid := 1, [35].log_data[7].valid := 1, [35].log_data[8].valid := 1, [35].log_data[9].valid := 1, [35].log_data[10].valid := 1, [35].log_data[11].valid := 1, [35].log_data[12].valid := 1, [35].log_data[13].valid := 1, [35].log_data[14].valid := 1, [35].log_data[15].valid := 1, [35].log_data[16].valid := 1, [35].log_data[17].valid := 1, [35].log_data[18].valid := 1, [35].log_data[19].valid := 1, [35].time.Year := 2023, [35].time.Month := 1, [35].time.Day := 16, [35].time.Hour := 9, [35].time.Minute := 14, [35].time.Second := 59, [36].log_data[0].min := 1.0, [36].log_data[0].max := 1.0, [36].log_data[0].total := 900.0, [36].log_data[0].time := 900.0, [36].log_data[0].minminute := 15, [36].log_data[0].maxminute := 15, [36].log_data[0].valid := 1, [36].log_data[1].valid := 1, [36].log_data[2].valid := 1,
        [36].log_data[3].valid := 1, [36].log_data[4].valid := 1, [36].log_data[5].valid := 1, [36].log_data[6].valid := 1, [36].log_data[7].valid := 1, [36].log_data[8].valid := 1, [36].log_data[9].valid := 1, [36].log_data[10].valid := 1, [36].log_data[11].valid := 1, [36].log_data[12].valid := 1, [36].log_data[13].valid := 1, [36].log_data[14].valid := 1, [36].log_data[15].valid := 1, [36].log_data[16].valid := 1, [36].log_data[17].valid := 1, [36].log_data[18].valid := 1, [36].log_data[19].valid := 1, [36].time.Year := 2023, [36].time.Month := 1, [36].time.Day := 16, [36].time.Hour := 9, [36].time.Minute := 29, [36].time.Second := 59, [37].log_data[0].min := 1.0, [37].log_data[0].max := 1.0, [37].log_data[0].total := 900.0, [37].log_data[0].time := 900.0, [37].log_data[0].minminute := 30, [37].log_data[0].maxminute := 30, [37].log_data[0].valid := 1, [37].log_data[1].valid := 1, [37].log_data[2].valid := 1, [37].log_data[3].valid := 1, [37].log_data[4].valid := 1, [37].log_data[5].valid := 1, [37].log_data[6].valid := 1, [37].log_data[7].valid := 1, [37].log_data[8].valid := 1, [37].log_data[9].valid := 1, [37].log_data[10].valid := 1, [37].log_data[11].valid := 1, [37].log_data[12].valid := 1, [37].log_data[13].valid := 1, [37].log_data[14].valid := 1, [37].log_data[15].valid := 1, [37].log_data[16].valid := 1, [37].log_data[17].valid := 1, [37].log_data[18].valid := 1, [37].log_data[19].valid := 1, [37].time.Year := 2023, [37].time.Month := 1, [37].time.Day := 16, [37].time.Hour := 9, [37].time.Minute := 44, [37].time.Second := 59, [38].log_data[0].min := 1.0, [38].log_data[0].max := 1.0, [38].log_data[0].total := 900.0, [38].log_data[0].time := 900.0, [38].log_data[0].minminute := 45,
        [38].log_data[0].maxminute := 45, [38].log_data[0].valid := 1, [38].log_data[1].valid := 1, [38].log_data[2].valid := 1, [38].log_data[3].valid := 1, [38].log_data[4].valid := 1, [38].log_data[5].valid := 1, [38].log_data[6].valid := 1, [38].log_data[7].valid := 1, [38].log_data[8].valid := 1, [38].log_data[9].valid := 1, [38].log_data[10].valid := 1, [38].log_data[11].valid := 1, [38].log_data[12].valid := 1, [38].log_data[13].valid := 1, [38].log_data[14].valid := 1, [38].log_data[15].valid := 1, [38].log_data[16].valid := 1, [38].log_data[17].valid := 1, [38].log_data[18].valid := 1, [38].log_data[19].valid := 1, [38].time.Year := 2023, [38].time.Month := 1, [38].time.Day := 16, [38].time.Hour := 9, [38].time.Minute := 59, [38].time.Second := 59, [39].log_data[0].min := 1.0, [39].log_data[0].max := 1.0, [39].log_data[0].total := 899.5, [39].log_data[0].time := 899.5, [39].log_data[0].valid := 1, [39].log_data[1].valid := 1, [39].log_data[2].valid := 1, [39].log_data[3].valid := 1, [39].log_data[4].valid := 1, [39].log_data[5].valid := 1, [39].log_data[6].valid := 1, [39].log_data[7].valid := 1, [39].log_data[8].valid := 1, [39].log_data[9].valid := 1, [39].log_data[10].valid := 1, [39].log_data[11].valid := 1, [39].log_data[12].valid := 1, [39].log_data[13].valid := 1, [39].log_data[14].valid := 1, [39].log_data[15].valid := 1, [39].log_data[16].valid := 1, [39].log_data[17].valid := 1, [39].log_data[18].valid := 1, [39].log_data[19].valid := 1, [39].time.Year := 2023, [39].time.Month := 1, [39].time.Day := 16, [39].time.Hour := 10, [39].time.Minute := 14, [39].time.Second := 59, [40].log_data[0].min := 1.0, [40].log_data[0].max := 1.0, [40].log_data[0].total := 900.0,
        [40].log_data[0].time := 900.0, [40].log_data[0].minminute := 15, [40].log_data[0].maxminute := 15, [40].log_data[0].valid := 1, [40].log_data[1].valid := 1, [40].log_data[2].valid := 1, [40].log_data[3].valid := 1, [40].log_data[4].valid := 1, [40].log_data[5].valid := 1, [40].log_data[6].valid := 1, [40].log_data[7].valid := 1, [40].log_data[8].valid := 1, [40].log_data[9].valid := 1, [40].log_data[10].valid := 1, [40].log_data[11].valid := 1, [40].log_data[12].valid := 1, [40].log_data[13].valid := 1, [40].log_data[14].valid := 1, [40].log_data[15].valid := 1, [40].log_data[16].valid := 1, [40].log_data[17].valid := 1, [40].log_data[18].valid := 1, [40].log_data[19].valid := 1, [40].time.Year := 2023, [40].time.Month := 1, [40].time.Day := 16, [40].time.Hour := 10, [40].time.Minute := 29, [40].time.Second := 59, [41].log_data[0].min := 1.0, [41].log_data[0].max := 1.0, [41].log_data[0].total := 900.0, [41].log_data[0].time := 900.0, [41].log_data[0].minminute := 30, [41].log_data[0].maxminute := 30, [41].log_data[0].valid := 1, [41].log_data[1].valid := 1, [41].log_data[2].valid := 1, [41].log_data[3].valid := 1, [41].log_data[4].valid := 1, [41].log_data[5].valid := 1, [41].log_data[6].valid := 1, [41].log_data[7].valid := 1, [41].log_data[8].valid := 1, [41].log_data[9].valid := 1, [41].log_data[10].valid := 1, [41].log_data[11].valid := 1, [41].log_data[12].valid := 1, [41].log_data[13].valid := 1, [41].log_data[14].valid := 1, [41].log_data[15].valid := 1, [41].log_data[16].valid := 1, [41].log_data[17].valid := 1, [41].log_data[18].valid := 1, [41].log_data[19].valid := 1, [41].time.Year := 2023, [41].time.Month := 1, [41].time.Day := 16, [41].time.Hour := 10, [41].time.Minute := 44,
        [41].time.Second := 59, [42].log_data[0].min := 1.0, [42].log_data[0].max := 1.0, [42].log_data[0].total := 900.0, [42].log_data[0].time := 900.0, [42].log_data[0].minminute := 45, [42].log_data[0].maxminute := 45, [42].log_data[0].valid := 1, [42].log_data[1].valid := 1, [42].log_data[2].valid := 1, [42].log_data[3].valid := 1, [42].log_data[4].valid := 1, [42].log_data[5].valid := 1, [42].log_data[6].valid := 1, [42].log_data[7].valid := 1, [42].log_data[8].valid := 1, [42].log_data[9].valid := 1, [42].log_data[10].valid := 1, [42].log_data[11].valid := 1, [42].log_data[12].valid := 1, [42].log_data[13].valid := 1, [42].log_data[14].valid := 1, [42].log_data[15].valid := 1, [42].log_data[16].valid := 1, [42].log_data[17].valid := 1, [42].log_data[18].valid := 1, [42].log_data[19].valid := 1, [42].time.Year := 2023, [42].time.Month := 1, [42].time.Day := 16, [42].time.Hour := 10, [42].time.Minute := 59, [42].time.Second := 59, [43].log_data[0].min := 1.0, [43].log_data[0].max := 1.0, [43].log_data[0].total := 900.0, [43].log_data[0].time := 900.0, [43].log_data[0].valid := 1, [43].log_data[1].valid := 1, [43].log_data[2].valid := 1, [43].log_data[3].valid := 1, [43].log_data[4].valid := 1, [43].log_data[5].valid := 1, [43].log_data[6].valid := 1, [43].log_data[7].valid := 1, [43].log_data[8].valid := 1, [43].log_data[9].valid := 1, [43].log_data[10].valid := 1, [43].log_data[11].valid := 1, [43].log_data[12].valid := 1, [43].log_data[13].valid := 1, [43].log_data[14].valid := 1, [43].log_data[15].valid := 1, [43].log_data[16].valid := 1, [43].log_data[17].valid := 1, [43].log_data[18].valid := 1, [43].log_data[19].valid := 1, [43].time.Year := 2023, [43].time.Month := 1, [43].time.Day := 16,
        [43].time.Hour := 11, [43].time.Minute := 14, [43].time.Second := 59, [44].log_data[0].min := 1.0, [44].log_data[0].max := 1.0, [44].log_data[0].total := 900.0, [44].log_data[0].time := 900.0, [44].log_data[0].minminute := 15, [44].log_data[0].maxminute := 15, [44].log_data[0].valid := 1, [44].log_data[1].valid := 1, [44].log_data[2].valid := 1, [44].log_data[3].valid := 1, [44].log_data[4].valid := 1, [44].log_data[5].valid := 1, [44].log_data[6].valid := 1, [44].log_data[7].valid := 1, [44].log_data[8].valid := 1, [44].log_data[9].valid := 1, [44].log_data[10].valid := 1, [44].log_data[11].valid := 1, [44].log_data[12].valid := 1, [44].log_data[13].valid := 1, [44].log_data[14].valid := 1, [44].log_data[15].valid := 1, [44].log_data[16].valid := 1, [44].log_data[17].valid := 1, [44].log_data[18].valid := 1, [44].log_data[19].valid := 1, [44].time.Year := 2023, [44].time.Month := 1, [44].time.Day := 16, [44].time.Hour := 11, [44].time.Minute := 29, [44].time.Second := 59, [45].log_data[0].min := 1.0, [45].log_data[0].max := 1.0, [45].log_data[0].total := 900.0, [45].log_data[0].time := 900.0, [45].log_data[0].minminute := 30, [45].log_data[0].maxminute := 30, [45].log_data[0].valid := 1, [45].log_data[1].valid := 1, [45].log_data[2].valid := 1, [45].log_data[3].valid := 1, [45].log_data[4].valid := 1, [45].log_data[5].valid := 1, [45].log_data[6].valid := 1, [45].log_data[7].valid := 1, [45].log_data[8].valid := 1, [45].log_data[9].valid := 1, [45].log_data[10].valid := 1, [45].log_data[11].valid := 1, [45].log_data[12].valid := 1, [45].log_data[13].valid := 1, [45].log_data[14].valid := 1, [45].log_data[15].valid := 1, [45].log_data[16].valid := 1, [45].log_data[17].valid := 1, [45].log_data[18].valid := 1,
        [45].log_data[19].valid := 1, [45].time.Year := 2023, [45].time.Month := 1, [45].time.Day := 16, [45].time.Hour := 11, [45].time.Minute := 44, [45].time.Second := 59, [46].log_data[0].min := 1.0, [46].log_data[0].max := 1.0, [46].log_data[0].total := 900.0, [46].log_data[0].time := 900.0, [46].log_data[0].minminute := 45, [46].log_data[0].maxminute := 45, [46].log_data[0].valid := 1, [46].log_data[1].valid := 1, [46].log_data[2].valid := 1, [46].log_data[3].valid := 1, [46].log_data[4].valid := 1, [46].log_data[5].valid := 1, [46].log_data[6].valid := 1, [46].log_data[7].valid := 1, [46].log_data[8].valid := 1, [46].log_data[9].valid := 1, [46].log_data[10].valid := 1, [46].log_data[11].valid := 1, [46].log_data[12].valid := 1, [46].log_data[13].valid := 1, [46].log_data[14].valid := 1, [46].log_data[15].valid := 1, [46].log_data[16].valid := 1, [46].log_data[17].valid := 1, [46].log_data[18].valid := 1, [46].log_data[19].valid := 1, [46].time.Year := 2023, [46].time.Month := 1, [46].time.Day := 16, [46].time.Hour := 11, [46].time.Minute := 59, [46].time.Second := 59, [47].log_data[0].min := 1.0, [47].log_data[0].max := 1.0, [47].log_data[0].total := 900.0, [47].log_data[0].time := 900.0, [47].log_data[0].valid := 1, [47].log_data[1].valid := 1, [47].log_data[2].valid := 1, [47].log_data[3].valid := 1, [47].log_data[4].valid := 1, [47].log_data[5].valid := 1, [47].log_data[6].valid := 1, [47].log_data[7].valid := 1, [47].log_data[8].valid := 1, [47].log_data[9].valid := 1, [47].log_data[10].valid := 1, [47].log_data[11].valid := 1, [47].log_data[12].valid := 1, [47].log_data[13].valid := 1, [47].log_data[14].valid := 1, [47].log_data[15].valid := 1, [47].log_data[16].valid := 1,
        [47].log_data[17].valid := 1, [47].log_data[18].valid := 1, [47].log_data[19].valid := 1, [47].time.Year := 2023, [47].time.Month := 1, [47].time.Day := 16, [47].time.Hour := 12, [47].time.Minute := 14, [47].time.Second := 59, [48].log_data[0].min := 1.0, [48].log_data[0].max := 1.0, [48].log_data[0].total := 900.0, [48].log_data[0].time := 900.0, [48].log_data[0].minminute := 15, [48].log_data[0].maxminute := 15, [48].log_data[0].valid := 1, [48].log_data[1].valid := 1, [48].log_data[2].valid := 1, [48].log_data[3].valid := 1, [48].log_data[4].valid := 1, [48].log_data[5].valid := 1, [48].log_data[6].valid := 1, [48].log_data[7].valid := 1, [48].log_data[8].valid := 1, [48].log_data[9].valid := 1, [48].log_data[10].valid := 1, [48].log_data[11].valid := 1, [48].log_data[12].valid := 1, [48].log_data[13].valid := 1, [48].log_data[14].valid := 1, [48].log_data[15].valid := 1, [48].log_data[16].valid := 1, [48].log_data[17].valid := 1, [48].log_data[18].valid := 1, [48].log_data[19].valid := 1, [48].time.Year := 2023, [48].time.Month := 1, [48].time.Day := 16, [48].time.Hour := 12, [48].time.Minute := 29, [48].time.Second := 59, [49].log_data[0].min := 1.0, [49].log_data[0].max := 1.0, [49].log_data[0].total := 900.0, [49].log_data[0].time := 900.0, [49].log_data[0].minminute := 30, [49].log_data[0].maxminute := 30, [49].log_data[0].valid := 1, [49].log_data[1].valid := 1, [49].log_data[2].valid := 1, [49].log_data[3].valid := 1, [49].log_data[4].valid := 1, [49].log_data[5].valid := 1, [49].log_data[6].valid := 1, [49].log_data[7].valid := 1, [49].log_data[8].valid := 1, [49].log_data[9].valid := 1, [49].log_data[10].valid := 1, [49].log_data[11].valid := 1, [49].log_data[12].valid := 1,
        [49].log_data[13].valid := 1, [49].log_data[14].valid := 1, [49].log_data[15].valid := 1, [49].log_data[16].valid := 1, [49].log_data[17].valid := 1, [49].log_data[18].valid := 1, [49].log_data[19].valid := 1, [49].time.Year := 2023, [49].time.Month := 1, [49].time.Day := 16, [49].time.Hour := 12, [49].time.Minute := 44, [49].time.Second := 59, [50].log_data[0].min := 1.0, [50].log_data[0].max := 1.0, [50].log_data[0].total := 900.0, [50].log_data[0].time := 900.0, [50].log_data[0].minminute := 45, [50].log_data[0].maxminute := 45, [50].log_data[0].valid := 1, [50].log_data[1].valid := 1, [50].log_data[2].valid := 1, [50].log_data[3].valid := 1, [50].log_data[4].valid := 1, [50].log_data[5].valid := 1, [50].log_data[6].valid := 1, [50].log_data[7].valid := 1, [50].log_data[8].valid := 1, [50].log_data[9].valid := 1, [50].log_data[10].valid := 1, [50].log_data[11].valid := 1, [50].log_data[12].valid := 1, [50].log_data[13].valid := 1, [50].log_data[14].valid := 1, [50].log_data[15].valid := 1, [50].log_data[16].valid := 1, [50].log_data[17].valid := 1, [50].log_data[18].valid := 1, [50].log_data[19].valid := 1, [50].time.Year := 2023, [50].time.Month := 1, [50].time.Day := 16, [50].time.Hour := 12, [50].time.Minute := 59, [50].time.Second := 59, [51].log_data[0].min := 1.0, [51].log_data[0].max := 1.0, [51].log_data[0].total := 900.0, [51].log_data[0].time := 900.0, [51].log_data[0].valid := 1, [51].log_data[1].valid := 1, [51].log_data[2].valid := 1, [51].log_data[3].valid := 1, [51].log_data[4].valid := 1, [51].log_data[5].valid := 1, [51].log_data[6].valid := 1, [51].log_data[7].valid := 1, [51].log_data[8].valid := 1, [51].log_data[9].valid := 1, [51].log_data[10].valid := 1,
        [51].log_data[11].valid := 1, [51].log_data[12].valid := 1, [51].log_data[13].valid := 1, [51].log_data[14].valid := 1, [51].log_data[15].valid := 1, [51].log_data[16].valid := 1, [51].log_data[17].valid := 1, [51].log_data[18].valid := 1, [51].log_data[19].valid := 1, [51].time.Year := 2023, [51].time.Month := 1, [51].time.Day := 16, [51].time.Hour := 13, [51].time.Minute := 14, [51].time.Second := 59, [52].log_data[0].min := 1.0, [52].log_data[0].max := 1.0, [52].log_data[0].total := 900.0, [52].log_data[0].time := 900.0, [52].log_data[0].minminute := 15, [52].log_data[0].maxminute := 15, [52].log_data[0].valid := 1, [52].log_data[1].valid := 1, [52].log_data[2].valid := 1, [52].log_data[3].valid := 1, [52].log_data[4].valid := 1, [52].log_data[5].valid := 1, [52].log_data[6].valid := 1, [52].log_data[7].valid := 1, [52].log_data[8].valid := 1, [52].log_data[9].valid := 1, [52].log_data[10].valid := 1, [52].log_data[11].valid := 1, [52].log_data[12].valid := 1, [52].log_data[13].valid := 1, [52].log_data[14].valid := 1, [52].log_data[15].valid := 1, [52].log_data[16].valid := 1, [52].log_data[17].valid := 1, [52].log_data[18].valid := 1, [52].log_data[19].valid := 1, [52].time.Year := 2023, [52].time.Month := 1, [52].time.Day := 16, [52].time.Hour := 13, [52].time.Minute := 29, [52].time.Second := 59, [53].log_data[0].min := 1.0, [53].log_data[0].max := 1.0, [53].log_data[0].total := 900.0, [53].log_data[0].time := 900.0, [53].log_data[0].minminute := 30, [53].log_data[0].maxminute := 30, [53].log_data[0].valid := 1, [53].log_data[1].valid := 1, [53].log_data[2].valid := 1, [53].log_data[3].valid := 1, [53].log_data[4].valid := 1, [53].log_data[5].valid := 1, [53].log_data[6].valid := 1,
        [53].log_data[7].valid := 1, [53].log_data[8].valid := 1, [53].log_data[9].valid := 1, [53].log_data[10].valid := 1, [53].log_data[11].valid := 1, [53].log_data[12].valid := 1, [53].log_data[13].valid := 1, [53].log_data[14].valid := 1, [53].log_data[15].valid := 1, [53].log_data[16].valid := 1, [53].log_data[17].valid := 1, [53].log_data[18].valid := 1, [53].log_data[19].valid := 1, [53].time.Year := 2023, [53].time.Month := 1, [53].time.Day := 16, [53].time.Hour := 13, [53].time.Minute := 44, [53].time.Second := 59, [54].log_data[0].min := 1.0, [54].log_data[0].max := 1.0, [54].log_data[0].total := 900.0, [54].log_data[0].time := 900.0, [54].log_data[0].minminute := 45, [54].log_data[0].maxminute := 45, [54].log_data[0].valid := 1, [54].log_data[1].valid := 1, [54].log_data[2].valid := 1, [54].log_data[3].valid := 1, [54].log_data[4].valid := 1, [54].log_data[5].valid := 1, [54].log_data[6].valid := 1, [54].log_data[7].valid := 1, [54].log_data[8].valid := 1, [54].log_data[9].valid := 1, [54].log_data[10].valid := 1, [54].log_data[11].valid := 1, [54].log_data[12].valid := 1, [54].log_data[13].valid := 1, [54].log_data[14].valid := 1, [54].log_data[15].valid := 1, [54].log_data[16].valid := 1, [54].log_data[17].valid := 1, [54].log_data[18].valid := 1, [54].log_data[19].valid := 1, [54].time.Year := 2023, [54].time.Month := 1, [54].time.Day := 16, [54].time.Hour := 13, [54].time.Minute := 59, [54].time.Second := 59, [55].log_data[0].min := 1.0, [55].log_data[0].max := 1.0, [55].log_data[0].total := 900.0, [55].log_data[0].time := 900.0, [55].log_data[0].valid := 1, [55].log_data[1].valid := 1, [55].log_data[2].valid := 1, [55].log_data[3].valid := 1, [55].log_data[4].valid := 1,
        [55].log_data[5].valid := 1, [55].log_data[6].valid := 1, [55].log_data[7].valid := 1, [55].log_data[8].valid := 1, [55].log_data[9].valid := 1, [55].log_data[10].valid := 1, [55].log_data[11].valid := 1, [55].log_data[12].valid := 1, [55].log_data[13].valid := 1, [55].log_data[14].valid := 1, [55].log_data[15].valid := 1, [55].log_data[16].valid := 1, [55].log_data[17].valid := 1, [55].log_data[18].valid := 1, [55].log_data[19].valid := 1, [55].time.Year := 2023, [55].time.Month := 1, [55].time.Day := 16, [55].time.Hour := 14, [55].time.Minute := 14, [55].time.Second := 59, [56].log_data[0].min := 1.0, [56].log_data[0].max := 1.0, [56].log_data[0].total := 900.0, [56].log_data[0].time := 900.0, [56].log_data[0].minminute := 15, [56].log_data[0].maxminute := 15, [56].log_data[0].valid := 1, [56].log_data[1].valid := 1, [56].log_data[2].valid := 1, [56].log_data[3].valid := 1, [56].log_data[4].valid := 1, [56].log_data[5].valid := 1, [56].log_data[6].valid := 1, [56].log_data[7].valid := 1, [56].log_data[8].valid := 1, [56].log_data[9].valid := 1, [56].log_data[10].valid := 1, [56].log_data[11].valid := 1, [56].log_data[12].valid := 1, [56].log_data[13].valid := 1, [56].log_data[14].valid := 1, [56].log_data[15].valid := 1, [56].log_data[16].valid := 1, [56].log_data[17].valid := 1, [56].log_data[18].valid := 1, [56].log_data[19].valid := 1, [56].time.Year := 2023, [56].time.Month := 1, [56].time.Day := 16, [56].time.Hour := 14, [56].time.Minute := 29, [56].time.Second := 59, [57].log_data[0].min := 1.0, [57].log_data[0].max := 1.0, [57].log_data[0].total := 900.0, [57].log_data[0].time := 900.0, [57].log_data[0].minminute := 30, [57].log_data[0].maxminute := 30, [57].log_data[0].valid := 1,
        [57].log_data[1].valid := 1, [57].log_data[2].valid := 1, [57].log_data[3].valid := 1, [57].log_data[4].valid := 1, [57].log_data[5].valid := 1, [57].log_data[6].valid := 1, [57].log_data[7].valid := 1, [57].log_data[8].valid := 1, [57].log_data[9].valid := 1, [57].log_data[10].valid := 1, [57].log_data[11].valid := 1, [57].log_data[12].valid := 1, [57].log_data[13].valid := 1, [57].log_data[14].valid := 1, [57].log_data[15].valid := 1, [57].log_data[16].valid := 1, [57].log_data[17].valid := 1, [57].log_data[18].valid := 1, [57].log_data[19].valid := 1, [57].time.Year := 2023, [57].time.Month := 1, [57].time.Day := 16, [57].time.Hour := 14, [57].time.Minute := 44, [57].time.Second := 59, [58].log_data[0].min := 1.0, [58].log_data[0].max := 1.0, [58].log_data[0].total := 900.0, [58].log_data[0].time := 900.0, [58].log_data[0].minminute := 45, [58].log_data[0].maxminute := 45, [58].log_data[0].valid := 1, [58].log_data[1].valid := 1, [58].log_data[2].valid := 1, [58].log_data[3].valid := 1, [58].log_data[4].valid := 1, [58].log_data[5].valid := 1, [58].log_data[6].valid := 1, [58].log_data[7].valid := 1, [58].log_data[8].valid := 1, [58].log_data[9].valid := 1, [58].log_data[10].valid := 1, [58].log_data[11].valid := 1, [58].log_data[12].valid := 1, [58].log_data[13].valid := 1, [58].log_data[14].valid := 1, [58].log_data[15].valid := 1, [58].log_data[16].valid := 1, [58].log_data[17].valid := 1, [58].log_data[18].valid := 1, [58].log_data[19].valid := 1, [58].time.Year := 2023, [58].time.Month := 1, [58].time.Day := 16, [58].time.Hour := 14, [58].time.Minute := 59, [58].time.Second := 59, [59].log_data[0].min := 1.0, [59].log_data[0].max := 1.0, [59].log_data[0].total := 900.0,
        [59].log_data[0].time := 900.0, [59].log_data[0].valid := 1, [59].log_data[1].valid := 1, [59].log_data[2].valid := 1, [59].log_data[3].valid := 1, [59].log_data[4].valid := 1, [59].log_data[5].valid := 1, [59].log_data[6].valid := 1, [59].log_data[7].valid := 1, [59].log_data[8].valid := 1, [59].log_data[9].valid := 1, [59].log_data[10].valid := 1, [59].log_data[11].valid := 1, [59].log_data[12].valid := 1, [59].log_data[13].valid := 1, [59].log_data[14].valid := 1, [59].log_data[15].valid := 1, [59].log_data[16].valid := 1, [59].log_data[17].valid := 1, [59].log_data[18].valid := 1, [59].log_data[19].valid := 1, [59].time.Year := 2023, [59].time.Month := 1, [59].time.Day := 16, [59].time.Hour := 15, [59].time.Minute := 14, [59].time.Second := 59, [60].log_data[0].min := 1.0, [60].log_data[0].max := 1.0, [60].log_data[0].total := 900.0, [60].log_data[0].time := 900.0, [60].log_data[0].minminute := 15, [60].log_data[0].maxminute := 15, [60].log_data[0].valid := 1, [60].log_data[1].valid := 1, [60].log_data[2].valid := 1, [60].log_data[3].valid := 1, [60].log_data[4].valid := 1, [60].log_data[5].valid := 1, [60].log_data[6].valid := 1, [60].log_data[7].valid := 1, [60].log_data[8].valid := 1, [60].log_data[9].valid := 1, [60].log_data[10].valid := 1, [60].log_data[11].valid := 1, [60].log_data[12].valid := 1, [60].log_data[13].valid := 1, [60].log_data[14].valid := 1, [60].log_data[15].valid := 1, [60].log_data[16].valid := 1, [60].log_data[17].valid := 1, [60].log_data[18].valid := 1, [60].log_data[19].valid := 1, [60].time.Year := 2023, [60].time.Month := 1, [60].time.Day := 16, [60].time.Hour := 15, [60].time.Minute := 29, [60].time.Second := 59, [61].log_data[0].min := 1.0,
        [61].log_data[0].max := 1.0, [61].log_data[0].total := 900.0, [61].log_data[0].time := 900.0, [61].log_data[0].minminute := 30, [61].log_data[0].maxminute := 30, [61].log_data[0].valid := 1, [61].log_data[1].valid := 1, [61].log_data[2].valid := 1, [61].log_data[3].valid := 1, [61].log_data[4].valid := 1, [61].log_data[5].valid := 1, [61].log_data[6].valid := 1, [61].log_data[7].valid := 1, [61].log_data[8].valid := 1, [61].log_data[9].valid := 1, [61].log_data[10].valid := 1, [61].log_data[11].valid := 1, [61].log_data[12].valid := 1, [61].log_data[13].valid := 1, [61].log_data[14].valid := 1, [61].log_data[15].valid := 1, [61].log_data[16].valid := 1, [61].log_data[17].valid := 1, [61].log_data[18].valid := 1, [61].log_data[19].valid := 1, [61].time.Year := 2023, [61].time.Month := 1, [61].time.Day := 16, [61].time.Hour := 15, [61].time.Minute := 44, [61].time.Second := 59, [62].log_data[0].min := 1.0, [62].log_data[0].max := 1.0, [62].log_data[0].total := 900.0, [62].log_data[0].time := 900.0, [62].log_data[0].minminute := 45, [62].log_data[0].maxminute := 45, [62].log_data[0].valid := 1, [62].log_data[1].valid := 1, [62].log_data[2].valid := 1, [62].log_data[3].valid := 1, [62].log_data[4].valid := 1, [62].log_data[5].valid := 1, [62].log_data[6].valid := 1, [62].log_data[7].valid := 1, [62].log_data[8].valid := 1, [62].log_data[9].valid := 1, [62].log_data[10].valid := 1, [62].log_data[11].valid := 1, [62].log_data[12].valid := 1, [62].log_data[13].valid := 1, [62].log_data[14].valid := 1, [62].log_data[15].valid := 1, [62].log_data[16].valid := 1, [62].log_data[17].valid := 1, [62].log_data[18].valid := 1, [62].log_data[19].valid := 1, [62].time.Year := 2023, [62].time.Month := 1, [62].time.Day := 16,
        [62].time.Hour := 15, [62].time.Minute := 59, [62].time.Second := 59, [63].log_data[0].min := 1.0, [63].log_data[0].max := 1.0, [63].log_data[0].total := 900.0, [63].log_data[0].time := 900.0, [63].log_data[0].valid := 1, [63].log_data[1].valid := 1, [63].log_data[2].valid := 1, [63].log_data[3].valid := 1, [63].log_data[4].valid := 1, [63].log_data[5].valid := 1, [63].log_data[6].valid := 1, [63].log_data[7].valid := 1, [63].log_data[8].valid := 1, [63].log_data[9].valid := 1, [63].log_data[10].valid := 1, [63].log_data[11].valid := 1, [63].log_data[12].valid := 1, [63].log_data[13].valid := 1, [63].log_data[14].valid := 1, [63].log_data[15].valid := 1, [63].log_data[16].valid := 1, [63].log_data[17].valid := 1, [63].log_data[18].valid := 1, [63].log_data[19].valid := 1, [63].time.Year := 2023, [63].time.Month := 1, [63].time.Day := 16, [63].time.Hour := 16, [63].time.Minute := 14, [63].time.Second := 59, [64].log_data[0].min := 1.0, [64].log_data[0].max := 1.0, [64].log_data[0].total := 900.0, [64].log_data[0].time := 900.0, [64].log_data[0].minminute := 15, [64].log_data[0].maxminute := 15, [64].log_data[0].valid := 1, [64].log_data[1].valid := 1, [64].log_data[2].valid := 1, [64].log_data[3].valid := 1, [64].log_data[4].valid := 1, [64].log_data[5].valid := 1, [64].log_data[6].valid := 1, [64].log_data[7].valid := 1, [64].log_data[8].valid := 1, [64].log_data[9].valid := 1, [64].log_data[10].valid := 1, [64].log_data[11].valid := 1, [64].log_data[12].valid := 1, [64].log_data[13].valid := 1, [64].log_data[14].valid := 1, [64].log_data[15].valid := 1, [64].log_data[16].valid := 1, [64].log_data[17].valid := 1, [64].log_data[18].valid := 1, [64].log_data[19].valid := 1, [64].time.Year := 2023,
        [64].time.Month := 1, [64].time.Day := 16, [64].time.Hour := 16, [64].time.Minute := 29, [64].time.Second := 59, [65].log_data[0].min := 1.0, [65].log_data[0].max := 1.0, [65].log_data[0].total := 900.0, [65].log_data[0].time := 900.0, [65].log_data[0].minminute := 30, [65].log_data[0].maxminute := 30, [65].log_data[0].valid := 1, [65].log_data[1].valid := 1, [65].log_data[2].valid := 1, [65].log_data[3].valid := 1, [65].log_data[4].valid := 1, [65].log_data[5].valid := 1, [65].log_data[6].valid := 1, [65].log_data[7].valid := 1, [65].log_data[8].valid := 1, [65].log_data[9].valid := 1, [65].log_data[10].valid := 1, [65].log_data[11].valid := 1, [65].log_data[12].valid := 1, [65].log_data[13].valid := 1, [65].log_data[14].valid := 1, [65].log_data[15].valid := 1, [65].log_data[16].valid := 1, [65].log_data[17].valid := 1, [65].log_data[18].valid := 1, [65].log_data[19].valid := 1, [65].time.Year := 2023, [65].time.Month := 1, [65].time.Day := 16, [65].time.Hour := 16, [65].time.Minute := 44, [65].time.Second := 59, [66].log_data[0].min := 1.0, [66].log_data[0].max := 1.0, [66].log_data[0].total := 900.0, [66].log_data[0].time := 900.0, [66].log_data[0].minminute := 45, [66].log_data[0].maxminute := 45, [66].log_data[0].valid := 1, [66].log_data[1].valid := 1, [66].log_data[2].valid := 1, [66].log_data[3].valid := 1, [66].log_data[4].valid := 1, [66].log_data[5].valid := 1, [66].log_data[6].valid := 1, [66].log_data[7].valid := 1, [66].log_data[8].valid := 1, [66].log_data[9].valid := 1, [66].log_data[10].valid := 1, [66].log_data[11].valid := 1, [66].log_data[12].valid := 1, [66].log_data[13].valid := 1, [66].log_data[14].valid := 1, [66].log_data[15].valid := 1, [66].log_data[16].valid := 1,
        [66].log_data[17].valid := 1, [66].log_data[18].valid := 1, [66].log_data[19].valid := 1, [66].time.Year := 2023, [66].time.Month := 1, [66].time.Day := 16, [66].time.Hour := 16, [66].time.Minute := 59, [66].time.Second := 59, [67].log_data[0].min := 1.0, [67].log_data[0].max := 1.0, [67].log_data[0].total := 900.0, [67].log_data[0].time := 900.0, [67].log_data[0].valid := 1, [67].log_data[1].valid := 1, [67].log_data[2].valid := 1, [67].log_data[3].valid := 1, [67].log_data[4].valid := 1, [67].log_data[5].valid := 1, [67].log_data[6].valid := 1, [67].log_data[7].valid := 1, [67].log_data[8].valid := 1, [67].log_data[9].valid := 1, [67].log_data[10].valid := 1, [67].log_data[11].valid := 1, [67].log_data[12].valid := 1, [67].log_data[13].valid := 1, [67].log_data[14].valid := 1, [67].log_data[15].valid := 1, [67].log_data[16].valid := 1, [67].log_data[17].valid := 1, [67].log_data[18].valid := 1, [67].log_data[19].valid := 1, [67].time.Year := 2023, [67].time.Month := 1, [67].time.Day := 16, [67].time.Hour := 17, [67].time.Minute := 14, [67].time.Second := 59, [68].log_data[0].min := 1.0, [68].log_data[0].max := 1.0, [68].log_data[0].total := 900.0, [68].log_data[0].time := 900.0, [68].log_data[0].minminute := 15, [68].log_data[0].maxminute := 15, [68].log_data[0].valid := 1, [68].log_data[1].valid := 1, [68].log_data[2].valid := 1, [68].log_data[3].valid := 1, [68].log_data[4].valid := 1, [68].log_data[5].valid := 1, [68].log_data[6].valid := 1, [68].log_data[7].valid := 1, [68].log_data[8].valid := 1, [68].log_data[9].valid := 1, [68].log_data[10].valid := 1, [68].log_data[11].valid := 1, [68].log_data[12].valid := 1, [68].log_data[13].valid := 1, [68].log_data[14].valid := 1,
        [68].log_data[15].valid := 1, [68].log_data[16].valid := 1, [68].log_data[17].valid := 1, [68].log_data[18].valid := 1, [68].log_data[19].valid := 1, [68].time.Year := 2023, [68].time.Month := 1, [68].time.Day := 16, [68].time.Hour := 17, [68].time.Minute := 29, [68].time.Second := 59, [69].log_data[0].min := 1.0, [69].log_data[0].max := 1.0, [69].log_data[0].total := 900.0, [69].log_data[0].time := 900.0, [69].log_data[0].minminute := 30, [69].log_data[0].maxminute := 30, [69].log_data[0].valid := 1, [69].log_data[1].valid := 1, [69].log_data[2].valid := 1, [69].log_data[3].valid := 1, [69].log_data[4].valid := 1, [69].log_data[5].valid := 1, [69].log_data[6].valid := 1, [69].log_data[7].valid := 1, [69].log_data[8].valid := 1, [69].log_data[9].valid := 1, [69].log_data[10].valid := 1, [69].log_data[11].valid := 1, [69].log_data[12].valid := 1, [69].log_data[13].valid := 1, [69].log_data[14].valid := 1, [69].log_data[15].valid := 1, [69].log_data[16].valid := 1, [69].log_data[17].valid := 1, [69].log_data[18].valid := 1, [69].log_data[19].valid := 1, [69].time.Year := 2023, [69].time.Month := 1, [69].time.Day := 16, [69].time.Hour := 17, [69].time.Minute := 44, [69].time.Second := 59, [70].log_data[0].min := 1.0, [70].log_data[0].max := 1.0, [70].log_data[0].total := 900.0, [70].log_data[0].time := 900.0, [70].log_data[0].minminute := 45, [70].log_data[0].maxminute := 45, [70].log_data[0].valid := 1, [70].log_data[1].valid := 1, [70].log_data[2].valid := 1, [70].log_data[3].valid := 1, [70].log_data[4].valid := 1, [70].log_data[5].valid := 1, [70].log_data[6].valid := 1, [70].log_data[7].valid := 1, [70].log_data[8].valid := 1, [70].log_data[9].valid := 1, [70].log_data[10].valid := 1,
        [70].log_data[11].valid := 1, [70].log_data[12].valid := 1, [70].log_data[13].valid := 1, [70].log_data[14].valid := 1, [70].log_data[15].valid := 1, [70].log_data[16].valid := 1, [70].log_data[17].valid := 1, [70].log_data[18].valid := 1, [70].log_data[19].valid := 1, [70].time.Year := 2023, [70].time.Month := 1, [70].time.Day := 16, [70].time.Hour := 17, [70].time.Minute := 59, [70].time.Second := 59, [71].log_data[0].min := 1.0, [71].log_data[0].max := 1.0, [71].log_data[0].total := 900.0, [71].log_data[0].time := 900.0, [71].log_data[0].valid := 1, [71].log_data[1].valid := 1, [71].log_data[2].valid := 1, [71].log_data[3].valid := 1, [71].log_data[4].valid := 1, [71].log_data[5].valid := 1, [71].log_data[6].valid := 1, [71].log_data[7].valid := 1, [71].log_data[8].valid := 1, [71].log_data[9].valid := 1, [71].log_data[10].valid := 1, [71].log_data[11].valid := 1, [71].log_data[12].valid := 1, [71].log_data[13].valid := 1, [71].log_data[14].valid := 1, [71].log_data[15].valid := 1, [71].log_data[16].valid := 1, [71].log_data[17].valid := 1, [71].log_data[18].valid := 1, [71].log_data[19].valid := 1, [71].time.Year := 2023, [71].time.Month := 1, [71].time.Day := 16, [71].time.Hour := 18, [71].time.Minute := 14, [71].time.Second := 59, [72].log_data[0].min := 1.0, [72].log_data[0].max := 1.0, [72].log_data[0].total := 900.0, [72].log_data[0].time := 900.0, [72].log_data[0].minminute := 15, [72].log_data[0].maxminute := 15, [72].log_data[0].valid := 1, [72].log_data[1].valid := 1, [72].log_data[2].valid := 1, [72].log_data[3].valid := 1, [72].log_data[4].valid := 1, [72].log_data[5].valid := 1, [72].log_data[6].valid := 1, [72].log_data[7].valid := 1, [72].log_data[8].valid := 1,
        [72].log_data[9].valid := 1, [72].log_data[10].valid := 1, [72].log_data[11].valid := 1, [72].log_data[12].valid := 1, [72].log_data[13].valid := 1, [72].log_data[14].valid := 1, [72].log_data[15].valid := 1, [72].log_data[16].valid := 1, [72].log_data[17].valid := 1, [72].log_data[18].valid := 1, [72].log_data[19].valid := 1, [72].time.Year := 2023, [72].time.Month := 1, [72].time.Day := 16, [72].time.Hour := 18, [72].time.Minute := 29, [72].time.Second := 59, [73].log_data[0].min := 1.0, [73].log_data[0].max := 1.0, [73].log_data[0].total := 900.0, [73].log_data[0].time := 900.0, [73].log_data[0].minminute := 30, [73].log_data[0].maxminute := 30, [73].log_data[0].valid := 1, [73].log_data[1].valid := 1, [73].log_data[2].valid := 1, [73].log_data[3].valid := 1, [73].log_data[4].valid := 1, [73].log_data[5].valid := 1, [73].log_data[6].valid := 1, [73].log_data[7].valid := 1, [73].log_data[8].valid := 1, [73].log_data[9].valid := 1, [73].log_data[10].valid := 1, [73].log_data[11].valid := 1, [73].log_data[12].valid := 1, [73].log_data[13].valid := 1, [73].log_data[14].valid := 1, [73].log_data[15].valid := 1, [73].log_data[16].valid := 1, [73].log_data[17].valid := 1, [73].log_data[18].valid := 1, [73].log_data[19].valid := 1, [73].time.Year := 2023, [73].time.Month := 1, [73].time.Day := 16, [73].time.Hour := 18, [73].time.Minute := 44, [73].time.Second := 59, [74].log_data[0].min := 1.0, [74].log_data[0].max := 1.0, [74].log_data[0].total := 900.0, [74].log_data[0].time := 900.0, [74].log_data[0].minminute := 45, [74].log_data[0].maxminute := 45, [74].log_data[0].valid := 1, [74].log_data[1].valid := 1, [74].log_data[2].valid := 1, [74].log_data[3].valid := 1, [74].log_data[4].valid := 1,
        [74].log_data[5].valid := 1, [74].log_data[6].valid := 1, [74].log_data[7].valid := 1, [74].log_data[8].valid := 1, [74].log_data[9].valid := 1, [74].log_data[10].valid := 1, [74].log_data[11].valid := 1, [74].log_data[12].valid := 1, [74].log_data[13].valid := 1, [74].log_data[14].valid := 1, [74].log_data[15].valid := 1, [74].log_data[16].valid := 1, [74].log_data[17].valid := 1, [74].log_data[18].valid := 1, [74].log_data[19].valid := 1, [74].time.Year := 2023, [74].time.Month := 1, [74].time.Day := 16, [74].time.Hour := 18, [74].time.Minute := 59, [74].time.Second := 59, [75].log_data[0].min := 1.0, [75].log_data[0].max := 1.0, [75].log_data[0].total := 900.0, [75].log_data[0].time := 900.0, [75].log_data[0].valid := 1, [75].log_data[1].valid := 1, [75].log_data[2].valid := 1, [75].log_data[3].valid := 1, [75].log_data[4].valid := 1, [75].log_data[5].valid := 1, [75].log_data[6].valid := 1, [75].log_data[7].valid := 1, [75].log_data[8].valid := 1, [75].log_data[9].valid := 1, [75].log_data[10].valid := 1, [75].log_data[11].valid := 1, [75].log_data[12].valid := 1, [75].log_data[13].valid := 1, [75].log_data[14].valid := 1, [75].log_data[15].valid := 1, [75].log_data[16].valid := 1, [75].log_data[17].valid := 1, [75].log_data[18].valid := 1, [75].log_data[19].valid := 1, [75].time.Year := 2023, [75].time.Month := 1, [75].time.Day := 16, [75].time.Hour := 19, [75].time.Minute := 14, [75].time.Second := 59, [76].log_data[0].min := 1.0, [76].log_data[0].max := 1.0, [76].log_data[0].total := 900.0, [76].log_data[0].time := 900.0, [76].log_data[0].minminute := 15, [76].log_data[0].maxminute := 15, [76].log_data[0].valid := 1, [76].log_data[1].valid := 1, [76].log_data[2].valid := 1,
        [76].log_data[3].valid := 1, [76].log_data[4].valid := 1, [76].log_data[5].valid := 1, [76].log_data[6].valid := 1, [76].log_data[7].valid := 1, [76].log_data[8].valid := 1, [76].log_data[9].valid := 1, [76].log_data[10].valid := 1, [76].log_data[11].valid := 1, [76].log_data[12].valid := 1, [76].log_data[13].valid := 1, [76].log_data[14].valid := 1, [76].log_data[15].valid := 1, [76].log_data[16].valid := 1, [76].log_data[17].valid := 1, [76].log_data[18].valid := 1, [76].log_data[19].valid := 1, [76].time.Year := 2023, [76].time.Month := 1, [76].time.Day := 16, [76].time.Hour := 19, [76].time.Minute := 29, [76].time.Second := 59, [77].log_data[0].min := 1.0, [77].log_data[0].max := 1.0, [77].log_data[0].total := 900.0, [77].log_data[0].time := 900.0, [77].log_data[0].minminute := 30, [77].log_data[0].maxminute := 30, [77].log_data[0].valid := 1, [77].log_data[1].valid := 1, [77].log_data[2].valid := 1, [77].log_data[3].valid := 1, [77].log_data[4].valid := 1, [77].log_data[5].valid := 1, [77].log_data[6].valid := 1, [77].log_data[7].valid := 1, [77].log_data[8].valid := 1, [77].log_data[9].valid := 1, [77].log_data[10].valid := 1, [77].log_data[11].valid := 1, [77].log_data[12].valid := 1, [77].log_data[13].valid := 1, [77].log_data[14].valid := 1, [77].log_data[15].valid := 1, [77].log_data[16].valid := 1, [77].log_data[17].valid := 1, [77].log_data[18].valid := 1, [77].log_data[19].valid := 1, [77].time.Year := 2023, [77].time.Month := 1, [77].time.Day := 16, [77].time.Hour := 19, [77].time.Minute := 44, [77].time.Second := 59, [78].log_data[0].min := 1.0, [78].log_data[0].max := 1.0, [78].log_data[0].total := 900.0, [78].log_data[0].time := 900.0, [78].log_data[0].minminute := 45,
        [78].log_data[0].maxminute := 45, [78].log_data[0].valid := 1, [78].log_data[1].valid := 1, [78].log_data[2].valid := 1, [78].log_data[3].valid := 1, [78].log_data[4].valid := 1, [78].log_data[5].valid := 1, [78].log_data[6].valid := 1, [78].log_data[7].valid := 1, [78].log_data[8].valid := 1, [78].log_data[9].valid := 1, [78].log_data[10].valid := 1, [78].log_data[11].valid := 1, [78].log_data[12].valid := 1, [78].log_data[13].valid := 1, [78].log_data[14].valid := 1, [78].log_data[15].valid := 1, [78].log_data[16].valid := 1, [78].log_data[17].valid := 1, [78].log_data[18].valid := 1, [78].log_data[19].valid := 1, [78].time.Year := 2023, [78].time.Month := 1, [78].time.Day := 16, [78].time.Hour := 19, [78].time.Minute := 59, [78].time.Second := 59, [79].log_data[0].min := 1.0, [79].log_data[0].max := 1.0, [79].log_data[0].total := 900.0, [79].log_data[0].time := 900.0, [79].log_data[0].valid := 1, [79].log_data[1].valid := 1, [79].log_data[2].valid := 1, [79].log_data[3].valid := 1, [79].log_data[4].valid := 1, [79].log_data[5].valid := 1, [79].log_data[6].valid := 1, [79].log_data[7].valid := 1, [79].log_data[8].valid := 1, [79].log_data[9].valid := 1, [79].log_data[10].valid := 1, [79].log_data[11].valid := 1, [79].log_data[12].valid := 1, [79].log_data[13].valid := 1, [79].log_data[14].valid := 1, [79].log_data[15].valid := 1, [79].log_data[16].valid := 1, [79].log_data[17].valid := 1, [79].log_data[18].valid := 1, [79].log_data[19].valid := 1, [79].time.Year := 2023, [79].time.Month := 1, [79].time.Day := 16, [79].time.Hour := 20, [79].time.Minute := 14, [79].time.Second := 59, [80].log_data[0].min := 1.0, [80].log_data[0].max := 1.0, [80].log_data[0].total := 900.0,
        [80].log_data[0].time := 900.0, [80].log_data[0].minminute := 15, [80].log_data[0].maxminute := 15, [80].log_data[0].valid := 1, [80].log_data[1].valid := 1, [80].log_data[2].valid := 1, [80].log_data[3].valid := 1, [80].log_data[4].valid := 1, [80].log_data[5].valid := 1, [80].log_data[6].valid := 1, [80].log_data[7].valid := 1, [80].log_data[8].valid := 1, [80].log_data[9].valid := 1, [80].log_data[10].valid := 1, [80].log_data[11].valid := 1, [80].log_data[12].valid := 1, [80].log_data[13].valid := 1, [80].log_data[14].valid := 1, [80].log_data[15].valid := 1, [80].log_data[16].valid := 1, [80].log_data[17].valid := 1, [80].log_data[18].valid := 1, [80].log_data[19].valid := 1, [80].time.Year := 2023, [80].time.Month := 1, [80].time.Day := 16, [80].time.Hour := 20, [80].time.Minute := 29, [80].time.Second := 59, [81].log_data[0].min := 1.0, [81].log_data[0].max := 1.0, [81].log_data[0].total := 900.0, [81].log_data[0].time := 900.0, [81].log_data[0].minminute := 30, [81].log_data[0].maxminute := 30, [81].log_data[0].valid := 1, [81].log_data[1].valid := 1, [81].log_data[2].valid := 1, [81].log_data[3].valid := 1, [81].log_data[4].valid := 1, [81].log_data[5].valid := 1, [81].log_data[6].valid := 1, [81].log_data[7].valid := 1, [81].log_data[8].valid := 1, [81].log_data[9].valid := 1, [81].log_data[10].valid := 1, [81].log_data[11].valid := 1, [81].log_data[12].valid := 1, [81].log_data[13].valid := 1, [81].log_data[14].valid := 1, [81].log_data[15].valid := 1, [81].log_data[16].valid := 1, [81].log_data[17].valid := 1, [81].log_data[18].valid := 1, [81].log_data[19].valid := 1, [81].time.Year := 2023, [81].time.Month := 1, [81].time.Day := 16, [81].time.Hour := 20, [81].time.Minute := 44,
        [81].time.Second := 59, [82].log_data[0].min := 1.0, [82].log_data[0].max := 1.0, [82].log_data[0].total := 900.0, [82].log_data[0].time := 900.0, [82].log_data[0].minminute := 45, [82].log_data[0].maxminute := 45, [82].log_data[0].valid := 1, [82].log_data[1].valid := 1, [82].log_data[2].valid := 1, [82].log_data[3].valid := 1, [82].log_data[4].valid := 1, [82].log_data[5].valid := 1, [82].log_data[6].valid := 1, [82].log_data[7].valid := 1, [82].log_data[8].valid := 1, [82].log_data[9].valid := 1, [82].log_data[10].valid := 1, [82].log_data[11].valid := 1, [82].log_data[12].valid := 1, [82].log_data[13].valid := 1, [82].log_data[14].valid := 1, [82].log_data[15].valid := 1, [82].log_data[16].valid := 1, [82].log_data[17].valid := 1, [82].log_data[18].valid := 1, [82].log_data[19].valid := 1, [82].time.Year := 2023, [82].time.Month := 1, [82].time.Day := 16, [82].time.Hour := 20, [82].time.Minute := 59, [82].time.Second := 59, [83].log_data[0].min := 1.0, [83].log_data[0].max := 1.0, [83].log_data[0].total := 899.5, [83].log_data[0].time := 899.5, [83].log_data[0].valid := 1, [83].log_data[1].valid := 1, [83].log_data[2].valid := 1, [83].log_data[3].valid := 1, [83].log_data[4].valid := 1, [83].log_data[5].valid := 1, [83].log_data[6].valid := 1, [83].log_data[7].valid := 1, [83].log_data[8].valid := 1, [83].log_data[9].valid := 1, [83].log_data[10].valid := 1, [83].log_data[11].valid := 1, [83].log_data[12].valid := 1, [83].log_data[13].valid := 1, [83].log_data[14].valid := 1, [83].log_data[15].valid := 1, [83].log_data[16].valid := 1, [83].log_data[17].valid := 1, [83].log_data[18].valid := 1, [83].log_data[19].valid := 1, [83].time.Year := 2023, [83].time.Month := 1, [83].time.Day := 16,
        [83].time.Hour := 21, [83].time.Minute := 14, [83].time.Second := 59, [84].log_data[0].min := 1.0, [84].log_data[0].max := 1.0, [84].log_data[0].total := 900.0, [84].log_data[0].time := 900.0, [84].log_data[0].minminute := 15, [84].log_data[0].maxminute := 15, [84].log_data[0].valid := 1, [84].log_data[1].valid := 1, [84].log_data[2].valid := 1, [84].log_data[3].valid := 1, [84].log_data[4].valid := 1, [84].log_data[5].valid := 1, [84].log_data[6].valid := 1, [84].log_data[7].valid := 1, [84].log_data[8].valid := 1, [84].log_data[9].valid := 1, [84].log_data[10].valid := 1, [84].log_data[11].valid := 1, [84].log_data[12].valid := 1, [84].log_data[13].valid := 1, [84].log_data[14].valid := 1, [84].log_data[15].valid := 1, [84].log_data[16].valid := 1, [84].log_data[17].valid := 1, [84].log_data[18].valid := 1, [84].log_data[19].valid := 1, [84].time.Year := 2023, [84].time.Month := 1, [84].time.Day := 16, [84].time.Hour := 21, [84].time.Minute := 29, [84].time.Second := 59, [85].log_data[0].min := 1.0, [85].log_data[0].max := 1.0, [85].log_data[0].total := 900.0, [85].log_data[0].time := 900.0, [85].log_data[0].minminute := 30, [85].log_data[0].maxminute := 30, [85].log_data[0].valid := 1, [85].log_data[1].valid := 1, [85].log_data[2].valid := 1, [85].log_data[3].valid := 1, [85].log_data[4].valid := 1, [85].log_data[5].valid := 1, [85].log_data[6].valid := 1, [85].log_data[7].valid := 1, [85].log_data[8].valid := 1, [85].log_data[9].valid := 1, [85].log_data[10].valid := 1, [85].log_data[11].valid := 1, [85].log_data[12].valid := 1, [85].log_data[13].valid := 1, [85].log_data[14].valid := 1, [85].log_data[15].valid := 1, [85].log_data[16].valid := 1, [85].log_data[17].valid := 1, [85].log_data[18].valid := 1,
        [85].log_data[19].valid := 1, [85].time.Year := 2023, [85].time.Month := 1, [85].time.Day := 16, [85].time.Hour := 21, [85].time.Minute := 44, [85].time.Second := 59, [86].log_data[0].min := 1.0, [86].log_data[0].max := 1.0, [86].log_data[0].total := 900.0, [86].log_data[0].time := 900.0, [86].log_data[0].minminute := 45, [86].log_data[0].maxminute := 45, [86].log_data[0].valid := 1, [86].log_data[1].valid := 1, [86].log_data[2].valid := 1, [86].log_data[3].valid := 1, [86].log_data[4].valid := 1, [86].log_data[5].valid := 1, [86].log_data[6].valid := 1, [86].log_data[7].valid := 1, [86].log_data[8].valid := 1, [86].log_data[9].valid := 1, [86].log_data[10].valid := 1, [86].log_data[11].valid := 1, [86].log_data[12].valid := 1, [86].log_data[13].valid := 1, [86].log_data[14].valid := 1, [86].log_data[15].valid := 1, [86].log_data[16].valid := 1, [86].log_data[17].valid := 1, [86].log_data[18].valid := 1, [86].log_data[19].valid := 1, [86].time.Year := 2023, [86].time.Month := 1, [86].time.Day := 16, [86].time.Hour := 21, [86].time.Minute := 59, [86].time.Second := 59, [87].log_data[0].min := 1.0, [87].log_data[0].max := 1.0, [87].log_data[0].total := 900.0, [87].log_data[0].time := 900.0, [87].log_data[0].valid := 1, [87].log_data[1].valid := 1, [87].log_data[2].valid := 1, [87].log_data[3].valid := 1, [87].log_data[4].valid := 1, [87].log_data[5].valid := 1, [87].log_data[6].valid := 1, [87].log_data[7].valid := 1, [87].log_data[8].valid := 1, [87].log_data[9].valid := 1, [87].log_data[10].valid := 1, [87].log_data[11].valid := 1, [87].log_data[12].valid := 1, [87].log_data[13].valid := 1, [87].log_data[14].valid := 1, [87].log_data[15].valid := 1, [87].log_data[16].valid := 1,
        [87].log_data[17].valid := 1, [87].log_data[18].valid := 1, [87].log_data[19].valid := 1, [87].time.Year := 2023, [87].time.Month := 1, [87].time.Day := 16, [87].time.Hour := 22, [87].time.Minute := 14, [87].time.Second := 59, [88].log_data[0].min := 1.0, [88].log_data[0].max := 1.0, [88].log_data[0].total := 900.0, [88].log_data[0].time := 900.0, [88].log_data[0].minminute := 15, [88].log_data[0].maxminute := 15, [88].log_data[0].valid := 1, [88].log_data[1].valid := 1, [88].log_data[2].valid := 1, [88].log_data[3].valid := 1, [88].log_data[4].valid := 1, [88].log_data[5].valid := 1, [88].log_data[6].valid := 1, [88].log_data[7].valid := 1, [88].log_data[8].valid := 1, [88].log_data[9].valid := 1, [88].log_data[10].valid := 1, [88].log_data[11].valid := 1, [88].log_data[12].valid := 1, [88].log_data[13].valid := 1, [88].log_data[14].valid := 1, [88].log_data[15].valid := 1, [88].log_data[16].valid := 1, [88].log_data[17].valid := 1, [88].log_data[18].valid := 1, [88].log_data[19].valid := 1, [88].time.Year := 2023, [88].time.Month := 1, [88].time.Day := 16, [88].time.Hour := 22, [88].time.Minute := 29, [88].time.Second := 59, [89].log_data[0].min := 1.0, [89].log_data[0].max := 1.0, [89].log_data[0].total := 900.0, [89].log_data[0].time := 900.0, [89].log_data[0].minminute := 30, [89].log_data[0].maxminute := 30, [89].log_data[0].valid := 1, [89].log_data[1].valid := 1, [89].log_data[2].valid := 1, [89].log_data[3].valid := 1, [89].log_data[4].valid := 1, [89].log_data[5].valid := 1, [89].log_data[6].valid := 1, [89].log_data[7].valid := 1, [89].log_data[8].valid := 1, [89].log_data[9].valid := 1, [89].log_data[10].valid := 1, [89].log_data[11].valid := 1, [89].log_data[12].valid := 1,
        [89].log_data[13].valid := 1, [89].log_data[14].valid := 1, [89].log_data[15].valid := 1, [89].log_data[16].valid := 1, [89].log_data[17].valid := 1, [89].log_data[18].valid := 1, [89].log_data[19].valid := 1, [89].time.Year := 2023, [89].time.Month := 1, [89].time.Day := 16, [89].time.Hour := 22, [89].time.Minute := 44, [89].time.Second := 59, [90].log_data[0].min := 1.0, [90].log_data[0].max := 1.0, [90].log_data[0].total := 900.0, [90].log_data[0].time := 900.0, [90].log_data[0].minminute := 45, [90].log_data[0].maxminute := 45, [90].log_data[0].valid := 1, [90].log_data[1].valid := 1, [90].log_data[2].valid := 1, [90].log_data[3].valid := 1, [90].log_data[4].valid := 1, [90].log_data[5].valid := 1, [90].log_data[6].valid := 1, [90].log_data[7].valid := 1, [90].log_data[8].valid := 1, [90].log_data[9].valid := 1, [90].log_data[10].valid := 1, [90].log_data[11].valid := 1, [90].log_data[12].valid := 1, [90].log_data[13].valid := 1, [90].log_data[14].valid := 1, [90].log_data[15].valid := 1, [90].log_data[16].valid := 1, [90].log_data[17].valid := 1, [90].log_data[18].valid := 1, [90].log_data[19].valid := 1, [90].time.Year := 2023, [90].time.Month := 1, [90].time.Day := 16, [90].time.Hour := 22, [90].time.Minute := 59, [90].time.Second := 59, [91].log_data[0].min := 1.0, [91].log_data[0].max := 1.0, [91].log_data[0].total := 900.0, [91].log_data[0].time := 900.0, [91].log_data[0].valid := 1, [91].log_data[1].valid := 1, [91].log_data[2].valid := 1, [91].log_data[3].valid := 1, [91].log_data[4].valid := 1, [91].log_data[5].valid := 1, [91].log_data[6].valid := 1, [91].log_data[7].valid := 1, [91].log_data[8].valid := 1, [91].log_data[9].valid := 1, [91].log_data[10].valid := 1,
        [91].log_data[11].valid := 1, [91].log_data[12].valid := 1, [91].log_data[13].valid := 1, [91].log_data[14].valid := 1, [91].log_data[15].valid := 1, [91].log_data[16].valid := 1, [91].log_data[17].valid := 1, [91].log_data[18].valid := 1, [91].log_data[19].valid := 1, [91].time.Year := 2023, [91].time.Month := 1, [91].time.Day := 16, [91].time.Hour := 23, [91].time.Minute := 14, [91].time.Second := 59, [92].log_data[0].min := 1.0, [92].log_data[0].max := 1.0, [92].log_data[0].total := 900.0, [92].log_data[0].time := 900.0, [92].log_data[0].minminute := 15, [92].log_data[0].maxminute := 15, [92].log_data[0].valid := 1, [92].log_data[1].valid := 1, [92].log_data[2].valid := 1, [92].log_data[3].valid := 1, [92].log_data[4].valid := 1, [92].log_data[5].valid := 1, [92].log_data[6].valid := 1, [92].log_data[7].valid := 1, [92].log_data[8].valid := 1, [92].log_data[9].valid := 1, [92].log_data[10].valid := 1, [92].log_data[11].valid := 1, [92].log_data[12].valid := 1, [92].log_data[13].valid := 1, [92].log_data[14].valid := 1, [92].log_data[15].valid := 1, [92].log_data[16].valid := 1, [92].log_data[17].valid := 1, [92].log_data[18].valid := 1, [92].log_data[19].valid := 1, [92].time.Year := 2023, [92].time.Month := 1, [92].time.Day := 16, [92].time.Hour := 23, [92].time.Minute := 29, [92].time.Second := 59, [93].log_data[0].min := 1.0, [93].log_data[0].max := 1.0, [93].log_data[0].total := 900.0, [93].log_data[0].time := 900.0, [93].log_data[0].minminute := 30, [93].log_data[0].maxminute := 30, [93].log_data[0].valid := 1, [93].log_data[1].valid := 1, [93].log_data[2].valid := 1, [93].log_data[3].valid := 1, [93].log_data[4].valid := 1, [93].log_data[5].valid := 1, [93].log_data[6].valid := 1,
